LIN {X 0,Y 458.337,Z 1107.303,A -85,B 0,C 180,E1 22685.631,E2 22685.631} C_VEL
LIN {X 0,Y 458.982,Z 1103.583,A -85,B 0,C 180,E1 22683.619,E2 22683.619} C_VEL
LIN {X 0,Y 459.798,Z 1098.163,A -85,B 0,C 180,E1 22681.742,E2 22681.742} C_VEL
LIN {X 0,Y 460.852,Z 1090.743,A -85,B 0,C 180,E1 22679.873,E2 22679.873} C_VEL
LIN {X 0,Y 461.948,Z 1082.306,A -85,B 0,C 180,E1 22678.261,E2 22678.261} C_VEL
LIN {X 0,Y 463.216,Z 1071.686,A -85,B 0,C 180,E1 22676.656,E2 22676.656} C_VEL
LIN {X 0,Y 464.446,Z 1059.795,A -85,B 0,C 180,E1 22675.243,E2 22675.243} C_VEL
LIN {X 0,Y 465.635,Z 1046.257,A -85,B 0,C 180,E1 22673.958,E2 22673.958} C_VEL
LIN {X 0,Y 466.68,Z 1031.493,A -85,B 0,C 180,E1 22672.859,E2 22672.859} C_VEL
LIN {X 0,Y 467.361,Z 1018.628,A -85,B 0,C 180,E1 22672.128,E2 22672.128} C_VEL
LIN {X 0,Y 467.859,Z 1006.332,A -85,B 0,C 180,E1 22671.572,E2 22671.572} C_VEL
LIN {X 0,Y 468.216,Z 991.858,A -85,B 0,C 180,E1 22671.079,E2 22671.079} C_VEL
LIN {X 0,Y 469.132,Z 950.411,A -85,B 0,C 180,E1 22670.184,E2 22670.184} C_VEL
LIN {X 0,Y 473.462,Z 851.354,A -85,B 0,C 180,E1 22668.053,E2 22668.053} C_VEL
LIN {X 0,Y 475.333,Z 822.809,A -85,B 0,C 180,E1 22665.625,E2 22665.625} C_VEL
LIN {X 0,Y 478.095,Z 777.566,A -85,B 0,C 180,E1 22661.778,E2 22661.778} C_VEL
LIN {X 0,Y 480.688,Z 736.093,A -85,B 0,C 180,E1 22658.266,E2 22658.266} C_VEL
LIN {X 0,Y 483.225,Z 700.221,A -85,B 0,C 180,E1 22655.232,E2 22655.232} C_VEL
LIN {X 0,Y 479.813,Z 688.191,A -85,B 0,C 180,E1 22653.642,E2 22653.642} C_VEL
LIN {X 0,Y 475.221,Z 675.87,A -85,B 0,C 180,E1 22651.742,E2 22651.742} C_VEL
LIN {X 0,Y 470.89,Z 666.546,A -85,B 0,C 180,E1 22650.032,E2 22650.032} C_VEL
LIN {X 0,Y 467.066,Z 658.908,A -85,B 0,C 180,E1 22648.429,E2 22648.429} C_VEL
LIN {X 0,Y 464.878,Z 654.816,A -85,B 0,C 180,E1 22647.468,E2 22647.468} C_VEL
LIN {X 0,Y 462.283,Z 651.075,A -85,B 0,C 180,E1 22646.376,E2 22646.376} C_VEL
LIN {X 0,Y 461.646,Z 649.194,A -85,B 0,C 180,E1 22645.937,E2 22645.937} C_VEL
LIN {X 0,Y 458.957,Z 646.06,A -85,B 0,C 180,E1 22644.734,E2 22644.734} C_VEL
LIN {X 0,Y 458.216,Z 643.592,A -85,B 0,C 180,E1 22644.093,E2 22644.093} C_VEL
LIN {X 0,Y 458.23,Z 643.587,A -85,B 0,C 180,E1 22640.374,E2 22640.374} C_VEL
LIN {X 0,Y 458.266,Z 643.803,A -85,B 0,C 180,E1 22637.145,E2 22637.145} C_VEL
LIN {X 0,Y 465.849,Z 666.114,A -85,B 0,C 180,E1 22633.489,E2 22633.489} C_VEL
LIN {X 0,Y 468.816,Z 675.017,A -85,B 0,C 180,E1 22632.146,E2 22632.146} C_VEL
LIN {X 0,Y 486.171,Z 709.362,A -85,B 0,C 180,E1 22629.877,E2 22629.877} C_VEL
LIN {X 0,Y 491.258,Z 720.243,A -85,B 0,C 180,E1 22629.242,E2 22629.242} C_VEL
LIN {X 0,Y 494.064,Z 737.412,A -85,B 0,C 180,E1 22628.646,E2 22628.646} C_VEL
LIN {X 0,Y 482.629,Z 981.186,A -85,B 0,C 180,E1 22624.108,E2 22624.108} C_VEL
LIN {X 0,Y 480.802,Z 1004.838,A -85,B 0,C 180,E1 22623.453,E2 22623.453} C_VEL
LIN {X 0,Y 478.769,Z 1026.444,A -85,B 0,C 180,E1 22622.64,E2 22622.64} C_VEL
LIN {X 0,Y 476.333,Z 1048.657,A -85,B 0,C 180,E1 22621.581,E2 22621.581} C_VEL
LIN {X 0,Y 473.788,Z 1069.533,A -85,B 0,C 180,E1 22620.351,E2 22620.351} C_VEL
LIN {X 0,Y 471.164,Z 1089.497,A -85,B 0,C 180,E1 22618.935,E2 22618.935} C_VEL
LIN {X 0,Y 468.474,Z 1108.558,A -85,B 0,C 180,E1 22617.313,E2 22617.313} C_VEL
LIN {X 0,Y 465.955,Z 1126.145,A -85,B 0,C 180,E1 22615.549,E2 22615.549} C_VEL
LIN {X 0,Y 463.62,Z 1142.393,A -85,B 0,C 180,E1 22613.648,E2 22613.648} C_VEL
LIN {X 0,Y 461.556,Z 1157.308,A -85,B 0,C 180,E1 22611.607,E2 22611.607} C_VEL
LIN {X 0,Y 459.786,Z 1170.792,A -85,B 0,C 180,E1 22609.432,E2 22609.432} C_VEL
LIN {X 0,Y 458.295,Z 1183.586,A -85,B 0,C 180,E1 22606.997,E2 22606.997} C_VEL
LIN {X 0,Y 457.241,Z 1194.282,A -85,B 0,C 180,E1 22604.563,E2 22604.563} C_VEL
LIN {X 0,Y 456.575,Z 1203.017,A -85,B 0,C 180,E1 22602.134,E2 22602.134} C_VEL
LIN {X 0,Y 456.199,Z 1210.324,A -85,B 0,C 180,E1 22599.587,E2 22599.587} C_VEL
LIN {X 0,Y 456.065,Z 1215.915,A -85,B 0,C 180,E1 22597.05,E2 22597.05} C_VEL
LIN {X 0,Y 456.056,Z 1219.591,A -85,B 0,C 180,E1 22594.651,E2 22594.651} C_VEL
LIN {X 0,Y 456.097,Z 1221.978,A -85,B 0,C 180,E1 22592.008,E2 22592.008} C_VEL
LIN {X 0,Y 456.094,Z 1222.654,A -85,B 0,C 180,E1 22589.621,E2 22589.621} C_VEL
LIN {X 0,Y 456.059,Z 1221.739,A -85,B 0,C 180,E1 22587.108,E2 22587.108} C_VEL
LIN {X 0,Y 456.022,Z 1219.335,A -85,B 0,C 180,E1 22584.588,E2 22584.588} C_VEL
LIN {X 0,Y 456.064,Z 1215.225,A -85,B 0,C 180,E1 22582.059,E2 22582.059} C_VEL
LIN {X 0,Y 456.309,Z 1209.17,A -85,B 0,C 180,E1 22579.392,E2 22579.392} C_VEL
LIN {X 0,Y 456.847,Z 1201.683,A -85,B 0,C 180,E1 22576.841,E2 22576.841} C_VEL
LIN {X 0,Y 457.781,Z 1192.207,A -85,B 0,C 180,E1 22574.284,E2 22574.284} C_VEL
LIN {X 0,Y 459.122,Z 1181.351,A -85,B 0,C 180,E1 22571.853,E2 22571.853} C_VEL
LIN {X 0,Y 460.874,Z 1169.238,A -85,B 0,C 180,E1 22569.554,E2 22569.554} C_VEL
LIN {X 0,Y 463.122,Z 1154.921,A -85,B 0,C 180,E1 22567.264,E2 22567.264} C_VEL
LIN {X 0,Y 465.787,Z 1139.175,A -85,B 0,C 180,E1 22565.117,E2 22565.117} C_VEL
LIN {X 0,Y 468.983,Z 1120.873,A -85,B 0,C 180,E1 22562.99,E2 22562.99} C_VEL
LIN {X 0,Y 472.427,Z 1101.443,A -85,B 0,C 180,E1 22561.081,E2 22561.081} C_VEL
LIN {X 0,Y 475.913,Z 1081.805,A -85,B 0,C 180,E1 22559.439,E2 22559.439} C_VEL
LIN {X 0,Y 479.703,Z 1059.729,A -85,B 0,C 180,E1 22557.89,E2 22557.89} C_VEL
LIN {X 0,Y 483.529,Z 1036.671,A -85,B 0,C 180,E1 22556.556,E2 22556.556} C_VEL
LIN {X 0,Y 487.071,Z 1014.04,A -85,B 0,C 180,E1 22555.486,E2 22555.486} C_VEL
LIN {X 0,Y 490.729,Z 988.982,A -85,B 0,C 180,E1 22554.548,E2 22554.548} C_VEL
LIN {X 0,Y 494.01,Z 962.501,A -85,B 0,C 180,E1 22553.788,E2 22553.788} C_VEL
LIN {X 0,Y 502.512,Z 886.864,A -85,B 0,C 180,E1 22551.886,E2 22551.886} C_VEL
LIN {X 0,Y 512.742,Z 815.166,A -85,B 0,C 180,E1 22550.007,E2 22550.007} C_VEL
LIN {X 0,Y 525.324,Z 742.891,A -85,B 0,C 180,E1 22548.094,E2 22548.094} C_VEL
LIN {X 0,Y 525.625,Z 739.764,A -85,B 0,C 180,E1 22547.895,E2 22547.895} C_VEL
LIN {X 0,Y 524.85,Z 735.088,A -85,B 0,C 180,E1 22546.983,E2 22546.983} C_VEL
LIN {X 0,Y 524.367,Z 731.897,A -85,B 0,C 180,E1 22546.122,E2 22546.122} C_VEL
LIN {X 0,Y 524.118,Z 729.55,A -85,B 0,C 180,E1 22545.057,E2 22545.057} C_VEL
LIN {X 0,Y 524.379,Z 728.32,A -85,B 0,C 180,E1 22544.038,E2 22544.038} C_VEL
LIN {X 0,Y 525.489,Z 728.89,A -85,B 0,C 180,E1 22542.575,E2 22542.575} C_VEL
LIN {X 0,Y 526.895,Z 731.802,A -85,B 0,C 180,E1 22541.405,E2 22541.405} C_VEL
LIN {X 0,Y 513.622,Z 804.551,A -85,B 0,C 180,E1 22539.481,E2 22539.481} C_VEL
LIN {X 0,Y 503.47,Z 872.417,A -85,B 0,C 180,E1 22537.696,E2 22537.696} C_VEL
LIN {X 0,Y 494.22,Z 950.824,A -85,B 0,C 180,E1 22535.659,E2 22535.659} C_VEL
LIN {X 0,Y 491.286,Z 974.469,A -85,B 0,C 180,E1 22534.814,E2 22534.814} C_VEL
LIN {X 0,Y 488.112,Z 997.009,A -85,B 0,C 180,E1 22533.793,E2 22533.793} C_VEL
LIN {X 0,Y 484.564,Z 1019.669,A -85,B 0,C 180,E1 22532.518,E2 22532.518} C_VEL
LIN {X 0,Y 480.93,Z 1040.911,A -85,B 0,C 180,E1 22531.064,E2 22531.064} C_VEL
LIN {X 0,Y 477.15,Z 1061.537,A -85,B 0,C 180,E1 22529.366,E2 22529.366} C_VEL
LIN {X 0,Y 473.79,Z 1078.913,A -85,B 0,C 180,E1 22527.667,E2 22527.667} C_VEL
LIN {X 0,Y 470.383,Z 1096.053,A -85,B 0,C 180,E1 22525.701,E2 22525.701} C_VEL
LIN {X 0,Y 467.258,Z 1111.645,A -85,B 0,C 180,E1 22523.591,E2 22523.591} C_VEL
LIN {X 0,Y 464.455,Z 1125.746,A -85,B 0,C 180,E1 22521.338,E2 22521.338} C_VEL
LIN {X 0,Y 462.024,Z 1138.267,A -85,B 0,C 180,E1 22518.945,E2 22518.945} C_VEL
LIN {X 0,Y 460.099,Z 1148.714,A -85,B 0,C 180,E1 22516.543,E2 22516.543} C_VEL
LIN {X 0,Y 458.529,Z 1158.219,A -85,B 0,C 180,E1 22513.881,E2 22513.881} C_VEL
LIN {X 0,Y 457.491,Z 1165.473,A -85,B 0,C 180,E1 22511.347,E2 22511.347} C_VEL
LIN {X 0,Y 456.811,Z 1170.96,A -85,B 0,C 180,E1 22508.816,E2 22508.816} C_VEL
LIN {X 0,Y 456.398,Z 1175.063,A -85,B 0,C 180,E1 22506.165,E2 22506.165} C_VEL
LIN {X 0,Y 456.205,Z 1177.569,A -85,B 0,C 180,E1 22503.521,E2 22503.521} C_VEL
LIN {X 0,Y 456.123,Z 1178.354,A -85,B 0,C 180,E1 22501.008,E2 22501.008} C_VEL
LIN {X 0,Y 456.09,Z 1177.621,A -85,B 0,C 180,E1 22498.37,E2 22498.37} C_VEL
LIN {X 0,Y 456.122,Z 1175.459,A -85,B 0,C 180,E1 22495.854,E2 22495.854} C_VEL
LIN {X 0,Y 456.255,Z 1171.659,A -85,B 0,C 180,E1 22493.333,E2 22493.333} C_VEL
LIN {X 0,Y 456.568,Z 1166.024,A -85,B 0,C 180,E1 22490.676,E2 22490.676} C_VEL
LIN {X 0,Y 457.13,Z 1158.966,A -85,B 0,C 180,E1 22488.138,E2 22488.138} C_VEL
LIN {X 0,Y 458.014,Z 1149.951,A -85,B 0,C 180,E1 22485.592,E2 22485.592} C_VEL
LIN {X 0,Y 459.234,Z 1139.531,A -85,B 0,C 180,E1 22483.17,E2 22483.17} C_VEL
LIN {X 0,Y 460.786,Z 1127.797,A -85,B 0,C 180,E1 22480.876,E2 22480.876} C_VEL
LIN {X 0,Y 462.67,Z 1114.375,A -85,B 0,C 180,E1 22478.664,E2 22478.664} C_VEL
LIN {X 0,Y 464.862,Z 1099.284,A -85,B 0,C 180,E1 22476.555,E2 22476.555} C_VEL
LIN {X 0,Y 467.373,Z 1082.277,A -85,B 0,C 180,E1 22474.533,E2 22474.533} C_VEL
LIN {X 0,Y 469.879,Z 1064.944,A -85,B 0,C 180,E1 22472.777,E2 22472.777} C_VEL
LIN {X 0,Y 472.502,Z 1046.063,A -85,B 0,C 180,E1 22471.156,E2 22471.156} C_VEL
LIN {X 0,Y 475.044,Z 1025.969,A -85,B 0,C 180,E1 22469.713,E2 22469.713} C_VEL
LIN {X 0,Y 477.5,Z 1004.905,A -85,B 0,C 180,E1 22468.46,E2 22468.46} C_VEL
LIN {X 0,Y 479.725,Z 983.049,A -85,B 0,C 180,E1 22467.402,E2 22467.402} C_VEL
LIN {X 0,Y 481.61,Z 960.789,A -85,B 0,C 180,E1 22466.551,E2 22466.551} C_VEL
LIN {X 0,Y 483.181,Z 937.605,A -85,B 0,C 180,E1 22465.897,E2 22465.897} C_VEL
LIN {X 0,Y 485.692,Z 881.128,A -85,B 0,C 180,E1 22464.823,E2 22464.823} C_VEL
LIN {X 0,Y 493.87,Z 706.895,A -85,B 0,C 180,E1 22461.609,E2 22461.609} C_VEL
LIN {X 0,Y 473.868,Z 671.342,A -85,B 0,C 180,E1 22459.2,E2 22459.2} C_VEL
LIN {X 0,Y 459.932,Z 647.609,A -85,B 0,C 180,E1 22457.384,E2 22457.384} C_VEL
LIN {X 0,Y 458.349,Z 644.303,A -85,B 0,C 180,E1 22457.157,E2 22457.157} C_VEL
LIN {X 0,Y 458.226,Z 643.591,A -85,B 0,C 180,E1 22457.098,E2 22457.098} C_VEL
LIN {X 0,Y 458.204,Z 643.595,A -85,B 0,C 180,E1 22453.397,E2 22453.397} C_VEL
LIN {X 0,Y 458.194,Z 643.592,A -85,B 0,C 180,E1 22449.818,E2 22449.818} C_VEL
LIN {X 0,Y 458.229,Z 643.588,A -85,B 0,C 180,E1 22446.099,E2 22446.099} C_VEL
LIN {X 0,Y 458.238,Z 643.584,A -85,B 0,C 180,E1 22442.394,E2 22442.394} C_VEL
LIN {X 0,Y 458.226,Z 643.59,A -85,B 0,C 180,E1 22438.691,E2 22438.691} C_VEL
LIN {X 0,Y 458.208,Z 643.593,A -85,B 0,C 180,E1 22435.047,E2 22435.047} C_VEL
LIN {X 0,Y 458.209,Z 643.589,A -85,B 0,C 180,E1 22431.508,E2 22431.508} C_VEL
LIN {X 0,Y 458.228,Z 643.582,A -85,B 0,C 180,E1 22427.789,E2 22427.789} C_VEL
LIN {X 0,Y 458.24,Z 643.579,A -85,B 0,C 180,E1 22424.147,E2 22424.147} C_VEL
LIN {X 0,Y 458.227,Z 643.59,A -85,B 0,C 180,E1 22420.436,E2 22420.436} C_VEL
LIN {X 0,Y 458.221,Z 643.588,A -85,B 0,C 180,E1 22416.769,E2 22416.769} C_VEL
LIN {X 0,Y 458.199,Z 643.579,A -85,B 0,C 180,E1 22413.004,E2 22413.004} C_VEL
LIN {X 0,Y 458.243,Z 643.589,A -85,B 0,C 180,E1 22409.252,E2 22409.252} C_VEL
LIN {X 0,Y 458.23,Z 643.574,A -85,B 0,C 180,E1 22405.496,E2 22405.496} C_VEL
LIN {X 0,Y 458.241,Z 643.586,A -85,B 0,C 180,E1 22402.552,E2 22402.552} C_VEL
LIN {X 0,Y 457.257,Z 643.71,A -85,B 0,C 180,E1 22401.59,E2 22401.59} C_VEL
LIN {X 0,Y 450.741,Z 644.5,A -85,B 0,C 180,E1 22398.81,E2 22398.81} C_VEL
LIN {X 0,Y 450.263,Z 644.562,A -85,B 0,C 180,E1 22398.173,E2 22398.173} C_VEL
LIN {X 0,Y 450.272,Z 644.581,A -85,B 0,C 180,E1 22394.512,E2 22394.512} C_VEL
LIN {X 0,Y 450.297,Z 644.578,A -85,B 0,C 180,E1 22390.816,E2 22390.816} C_VEL
LIN {X 0,Y 450.3,Z 644.576,A -85,B 0,C 180,E1 22387.136,E2 22387.136} C_VEL
LIN {X 0,Y 450.282,Z 644.581,A -85,B 0,C 180,E1 22383.351,E2 22383.351} C_VEL
LIN {X 0,Y 450.266,Z 644.582,A -85,B 0,C 180,E1 22379.732,E2 22379.732} C_VEL
LIN {X 0,Y 450.271,Z 644.582,A -85,B 0,C 180,E1 22375.975,E2 22375.975} C_VEL
LIN {X 0,Y 450.303,Z 644.577,A -85,B 0,C 180,E1 22372.207,E2 22372.207} C_VEL
LIN {X 0,Y 450.293,Z 644.577,A -85,B 0,C 180,E1 22368.439,E2 22368.439} C_VEL
LIN {X 0,Y 450.313,Z 644.69,A -85,B 0,C 180,E1 22367.619,E2 22367.619} C_VEL
LIN {X 0,Y 458.281,Z 670.797,A -85,B 0,C 180,E1 22364.754,E2 22364.754} C_VEL
LIN {X 0,Y 463.683,Z 690.602,A -85,B 0,C 180,E1 22362.668,E2 22362.668} C_VEL
LIN {X 0,Y 461.849,Z 733.114,A -85,B 0,C 180,E1 22358.997,E2 22358.997} C_VEL
LIN {X 0,Y 460.019,Z 774.082,A -85,B 0,C 180,E1 22355.471,E2 22355.471} C_VEL
LIN {X 0,Y 458.233,Z 816.759,A -85,B 0,C 180,E1 22351.8,E2 22351.8} C_VEL
LIN {X 0,Y 457.335,Z 841.237,A -85,B 0,C 180,E1 22349.747,E2 22349.747} C_VEL
LIN {X 0,Y 454.489,Z 984.58,A -85,B 0,C 180,E1 22346.943,E2 22346.943} C_VEL
LIN {X 0,Y 454.254,Z 1000.505,A -85,B 0,C 180,E1 22346.432,E2 22346.432} C_VEL
LIN {X 0,Y 453.773,Z 1017.239,A -85,B 0,C 180,E1 22345.654,E2 22345.654} C_VEL
LIN {X 0,Y 453.21,Z 1032.259,A -85,B 0,C 180,E1 22344.71,E2 22344.71} C_VEL
LIN {X 0,Y 452.517,Z 1047.114,A -85,B 0,C 180,E1 22343.516,E2 22343.516} C_VEL
LIN {X 0,Y 451.77,Z 1060.968,A -85,B 0,C 180,E1 22342.099,E2 22342.099} C_VEL
LIN {X 0,Y 451.111,Z 1072.473,A -85,B 0,C 180,E1 22340.632,E2 22340.632} C_VEL
LIN {X 0,Y 450.49,Z 1083.338,A -85,B 0,C 180,E1 22338.905,E2 22338.905} C_VEL
LIN {X 0,Y 450.048,Z 1091.85,A -85,B 0,C 180,E1 22337.184,E2 22337.184} C_VEL
LIN {X 0,Y 449.732,Z 1099.321,A -85,B 0,C 180,E1 22335.233,E2 22335.233} C_VEL
LIN {X 0,Y 449.564,Z 1104.421,A -85,B 0,C 180,E1 22333.371,E2 22333.371} C_VEL
LIN {X 0,Y 449.564,Z 1108.099,A -85,B 0,C 180,E1 22331.414,E2 22331.414} C_VEL
LIN {X 0,Y 449.693,Z 1109.939,A -85,B 0,C 180,E1 22329.467,E2 22329.467} C_VEL
LIN {X 0,Y 450.004,Z 1110.041,A -85,B 0,C 180,E1 22327.402,E2 22327.402} C_VEL
LIN {X 0,Y 450.468,Z 1108.36,A -85,B 0,C 180,E1 22325.474,E2 22325.474} C_VEL
LIN {X 0,Y 451.167,Z 1104.684,A -85,B 0,C 180,E1 22323.428,E2 22323.428} C_VEL
LIN {X 0,Y 452.05,Z 1099.312,A -85,B 0,C 180,E1 22321.518,E2 22321.518} C_VEL
LIN {X 0,Y 453.175,Z 1091.901,A -85,B 0,C 180,E1 22319.618,E2 22319.618} C_VEL
LIN {X 0,Y 454.34,Z 1083.471,A -85,B 0,C 180,E1 22317.979,E2 22317.979} C_VEL
LIN {X 0,Y 455.686,Z 1072.872,A -85,B 0,C 180,E1 22316.349,E2 22316.349} C_VEL
LIN {X 0,Y 457.004,Z 1061.08,A -85,B 0,C 180,E1 22314.914,E2 22314.914} C_VEL
LIN {X 0,Y 458.218,Z 1048.37,A -85,B 0,C 180,E1 22313.671,E2 22313.671} C_VEL
LIN {X 0,Y 459.312,Z 1033.812,A -85,B 0,C 180,E1 22312.555,E2 22312.555} C_VEL
LIN {X 0,Y 460.035,Z 1021.306,A -85,B 0,C 180,E1 22311.813,E2 22311.813} C_VEL
LIN {X 0,Y 460.598,Z 1008.702,A -85,B 0,C 180,E1 22311.218,E2 22311.218} C_VEL
LIN {X 0,Y 461.027,Z 993.799,A -85,B 0,C 180,E1 22310.685,E2 22310.685} C_VEL
LIN {X 0,Y 461.915,Z 955.217,A -85,B 0,C 180,E1 22309.813,E2 22309.813} C_VEL
LIN {X 0,Y 466.569,Z 853.052,A -85,B 0,C 180,E1 22307.576,E2 22307.576} C_VEL
LIN {X 0,Y 467.129,Z 848.404,A -85,B 0,C 180,E1 22307.198,E2 22307.198} C_VEL
LIN {X 0,Y 470.047,Z 802.606,A -85,B 0,C 180,E1 22303.245,E2 22303.245} C_VEL
LIN {X 0,Y 472.898,Z 759.889,A -85,B 0,C 180,E1 22299.579,E2 22299.579} C_VEL
LIN {X 0,Y 476.042,Z 716.875,A -85,B 0,C 180,E1 22295.885,E2 22295.885} C_VEL
LIN {X 0,Y 477.044,Z 703.66,A -85,B 0,C 180,E1 22294.75,E2 22294.75} C_VEL
LIN {X 0,Y 473.589,Z 691.406,A -85,B 0,C 180,E1 22293.063,E2 22293.063} C_VEL
LIN {X 0,Y 469.425,Z 680.099,A -85,B 0,C 180,E1 22291.222,E2 22291.222} C_VEL
LIN {X 0,Y 464.623,Z 669.452,A -85,B 0,C 180,E1 22289.162,E2 22289.162} C_VEL
LIN {X 0,Y 462.016,Z 664.602,A -85,B 0,C 180,E1 22288.029,E2 22288.029} C_VEL
LIN {X 0,Y 459.954,Z 660.63,A -85,B 0,C 180,E1 22287.043,E2 22287.043} C_VEL
LIN {X 0,Y 457.831,Z 657.042,A -85,B 0,C 180,E1 22286.004,E2 22286.004} C_VEL
LIN {X 0,Y 457.236,Z 655.752,A -85,B 0,C 180,E1 22285.651,E2 22285.651} C_VEL
LIN {X 0,Y 454.733,Z 652.236,A -85,B 0,C 180,E1 22284.357,E2 22284.357} C_VEL
LIN {X 0,Y 454.056,Z 650.421,A -85,B 0,C 180,E1 22283.828,E2 22283.828} C_VEL
LIN {X 0,Y 451.212,Z 647.452,A -85,B 0,C 180,E1 22282.13,E2 22282.13} C_VEL
LIN {X 0,Y 450.294,Z 644.579,A -85,B 0,C 180,E1 22281,E2 22281} C_VEL
LIN {X 0,Y 450.298,Z 644.624,A -85,B 0,C 180,E1 22277.807,E2 22277.807} C_VEL
LIN {X 0,Y 457.888,Z 666.977,A -85,B 0,C 180,E1 22274.072,E2 22274.072} C_VEL
LIN {X 0,Y 460.437,Z 674.616,A -85,B 0,C 180,E1 22272.889,E2 22272.889} C_VEL
LIN {X 0,Y 477.823,Z 708.748,A -85,B 0,C 180,E1 22270.568,E2 22270.568} C_VEL
LIN {X 0,Y 484.83,Z 723.669,A -85,B 0,C 180,E1 22269.653,E2 22269.653} C_VEL
LIN {X 0,Y 487.245,Z 738.83,A -85,B 0,C 180,E1 22269.123,E2 22269.123} C_VEL
LIN {X 0,Y 475.415,Z 980.893,A -85,B 0,C 180,E1 22264.525,E2 22264.525} C_VEL
LIN {X 0,Y 473.536,Z 1004.519,A -85,B 0,C 180,E1 22263.86,E2 22263.86} C_VEL
LIN {X 0,Y 471.377,Z 1026.768,A -85,B 0,C 180,E1 22263.007,E2 22263.007} C_VEL
LIN {X 0,Y 468.865,Z 1048.922,A -85,B 0,C 180,E1 22261.927,E2 22261.927} C_VEL
LIN {X 0,Y 466.265,Z 1069.575,A -85,B 0,C 180,E1 22260.687,E2 22260.687} C_VEL
LIN {X 0,Y 463.558,Z 1089.559,A -85,B 0,C 180,E1 22259.243,E2 22259.243} C_VEL
LIN {X 0,Y 460.796,Z 1108.578,A -85,B 0,C 180,E1 22257.596,E2 22257.596} C_VEL
LIN {X 0,Y 458.208,Z 1126.129,A -85,B 0,C 180,E1 22255.805,E2 22255.805} C_VEL
LIN {X 0,Y 455.729,Z 1142.879,A -85,B 0,C 180,E1 22253.802,E2 22253.802} C_VEL
LIN {X 0,Y 453.626,Z 1157.705,A -85,B 0,C 180,E1 22251.732,E2 22251.732} C_VEL
LIN {X 0,Y 451.778,Z 1171.427,A -85,B 0,C 180,E1 22249.462,E2 22249.462} C_VEL
LIN {X 0,Y 450.301,Z 1183.795,A -85,B 0,C 180,E1 22247.042,E2 22247.042} C_VEL
LIN {X 0,Y 449.235,Z 1194.392,A -85,B 0,C 180,E1 22244.565,E2 22244.565} C_VEL
LIN {X 0,Y 448.564,Z 1203.082,A -85,B 0,C 180,E1 22242.093,E2 22242.093} C_VEL
LIN {X 0,Y 448.202,Z 1210.109,A -85,B 0,C 180,E1 22239.571,E2 22239.571} C_VEL
LIN {X 0,Y 448.073,Z 1215.549,A -85,B 0,C 180,E1 22237.048,E2 22237.048} C_VEL
LIN {X 0,Y 448.068,Z 1219.215,A -85,B 0,C 180,E1 22234.606,E2 22234.606} C_VEL
LIN {X 0,Y 448.11,Z 1221.575,A -85,B 0,C 180,E1 22231.916,E2 22231.916} C_VEL
LIN {X 0,Y 448.104,Z 1222.229,A -85,B 0,C 180,E1 22229.487,E2 22229.487} C_VEL
LIN {X 0,Y 448.062,Z 1221.271,A -85,B 0,C 180,E1 22226.928,E2 22226.928} C_VEL
LIN {X 0,Y 448.023,Z 1218.823,A -85,B 0,C 180,E1 22224.363,E2 22224.363} C_VEL
LIN {X 0,Y 448.083,Z 1214.671,A -85,B 0,C 180,E1 22221.788,E2 22221.788} C_VEL
LIN {X 0,Y 448.361,Z 1208.565,A -85,B 0,C 180,E1 22219.071,E2 22219.071} C_VEL
LIN {X 0,Y 448.964,Z 1201.029,A -85,B 0,C 180,E1 22216.475,E2 22216.475} C_VEL
LIN {X 0,Y 449.989,Z 1191.515,A -85,B 0,C 180,E1 22213.872,E2 22213.872} C_VEL
LIN {X 0,Y 451.451,Z 1180.617,A -85,B 0,C 180,E1 22211.4,E2 22211.4} C_VEL
LIN {X 0,Y 453.468,Z 1167.711,A -85,B 0,C 180,E1 22208.934,E2 22208.934} C_VEL
LIN {X 0,Y 455.924,Z 1153.321,A -85,B 0,C 180,E1 22206.611,E2 22206.611} C_VEL
LIN {X 0,Y 458.888,Z 1136.937,A -85,B 0,C 180,E1 22204.371,E2 22204.371} C_VEL
LIN {X 0,Y 462.147,Z 1119.572,A -85,B 0,C 180,E1 22202.347,E2 22202.347} C_VEL
LIN {X 0,Y 465.834,Z 1100.126,A -85,B 0,C 180,E1 22200.416,E2 22200.416} C_VEL
LIN {X 0,Y 469.684,Z 1079.787,A -85,B 0,C 180,E1 22198.704,E2 22198.704} C_VEL
LIN {X 0,Y 473.774,Z 1057.66,A -85,B 0,C 180,E1 22197.14,E2 22197.14} C_VEL
LIN {X 0,Y 478.026,Z 1033.867,A -85,B 0,C 180,E1 22195.758,E2 22195.758} C_VEL
LIN {X 0,Y 482.157,Z 1009.227,A -85,B 0,C 180,E1 22194.601,E2 22194.601} C_VEL
LIN {X 0,Y 486.308,Z 982.698,A -85,B 0,C 180,E1 22193.639,E2 22193.639} C_VEL
LIN {X 0,Y 490.024,Z 953.283,A -85,B 0,C 180,E1 22192.82,E2 22192.82} C_VEL
LIN {X 0,Y 498.645,Z 884.788,A -85,B 0,C 180,E1 22191.04,E2 22191.04} C_VEL
LIN {X 0,Y 509.832,Z 813.836,A -85,B 0,C 180,E1 22189.136,E2 22189.136} C_VEL
LIN {X 0,Y 522.832,Z 745.199,A -85,B 0,C 180,E1 22187.29,E2 22187.29} C_VEL
LIN {X 0,Y 522.275,Z 739.861,A -85,B 0,C 180,E1 22186.088,E2 22186.088} C_VEL
LIN {X 0,Y 522.1,Z 737.122,A -85,B 0,C 180,E1 22184.878,E2 22184.878} C_VEL
LIN {X 0,Y 522.417,Z 736.065,A -85,B 0,C 180,E1 22183.973,E2 22183.973} C_VEL
LIN {X 0,Y 523.403,Z 736.623,A -85,B 0,C 180,E1 22182.65,E2 22182.65} C_VEL
LIN {X 0,Y 523.881,Z 737.963,A -85,B 0,C 180,E1 22182.109,E2 22182.109} C_VEL
LIN {X 0,Y 509.719,Z 810.287,A -85,B 0,C 180,E1 22180.174,E2 22180.174} C_VEL
LIN {X 0,Y 498.675,Z 878.354,A -85,B 0,C 180,E1 22178.342,E2 22178.342} C_VEL
LIN {X 0,Y 489.185,Z 951.63,A -85,B 0,C 180,E1 22176.378,E2 22176.378} C_VEL
LIN {X 0,Y 486.052,Z 974.778,A -85,B 0,C 180,E1 22175.534,E2 22175.534} C_VEL
LIN {X 0,Y 482.482,Z 997.964,A -85,B 0,C 180,E1 22174.457,E2 22174.457} C_VEL
LIN {X 0,Y 478.713,Z 1020.215,A -85,B 0,C 180,E1 22173.18,E2 22173.18} C_VEL
LIN {X 0,Y 474.796,Z 1041.439,A -85,B 0,C 180,E1 22171.7,E2 22171.7} C_VEL
LIN {X 0,Y 470.962,Z 1060.961,A -85,B 0,C 180,E1 22170.072,E2 22170.072} C_VEL
LIN {X 0,Y 467.253,Z 1078.976,A -85,B 0,C 180,E1 22168.296,E2 22168.296} C_VEL
LIN {X 0,Y 463.519,Z 1096.576,A -85,B 0,C 180,E1 22166.248,E2 22166.248} C_VEL
LIN {X 0,Y 460.252,Z 1111.837,A -85,B 0,C 180,E1 22164.153,E2 22164.153} C_VEL
LIN {X 0,Y 457.35,Z 1125.463,A -85,B 0,C 180,E1 22161.956,E2 22161.956} C_VEL
LIN {X 0,Y 454.706,Z 1138.037,A -85,B 0,C 180,E1 22159.529,E2 22159.529} C_VEL
LIN {X 0,Y 452.617,Z 1148.6,A -85,B 0,C 180,E1 22157.089,E2 22157.089} C_VEL
LIN {X 0,Y 450.951,Z 1157.821,A -85,B 0,C 180,E1 22154.513,E2 22154.513} C_VEL
LIN {X 0,Y 449.713,Z 1165.568,A -85,B 0,C 180,E1 22151.806,E2 22151.806} C_VEL
LIN {X 0,Y 448.912,Z 1171.367,A -85,B 0,C 180,E1 22149.102,E2 22149.102} C_VEL
LIN {X 0,Y 448.452,Z 1175.481,A -85,B 0,C 180,E1 22146.403,E2 22146.403} C_VEL
LIN {X 0,Y 448.235,Z 1177.933,A -85,B 0,C 180,E1 22143.84,E2 22143.84} C_VEL
LIN {X 0,Y 448.138,Z 1178.782,A -85,B 0,C 180,E1 22141.153,E2 22141.153} C_VEL
LIN {X 0,Y 448.1,Z 1178.058,A -85,B 0,C 180,E1 22138.468,E2 22138.468} C_VEL
LIN {X 0,Y 448.13,Z 1175.827,A -85,B 0,C 180,E1 22135.852,E2 22135.852} C_VEL
LIN {X 0,Y 448.263,Z 1172.08,A -85,B 0,C 180,E1 22133.342,E2 22133.342} C_VEL
LIN {X 0,Y 448.584,Z 1166.432,A -85,B 0,C 180,E1 22130.638,E2 22130.638} C_VEL
LIN {X 0,Y 449.164,Z 1159.356,A -85,B 0,C 180,E1 22128.055,E2 22128.055} C_VEL
LIN {X 0,Y 450.077,Z 1150.31,A -85,B 0,C 180,E1 22125.464,E2 22125.464} C_VEL
LIN {X 0,Y 451.34,Z 1139.852,A -85,B 0,C 180,E1 22123,E2 22123} C_VEL
LIN {X 0,Y 452.946,Z 1128.076,A -85,B 0,C 180,E1 22120.666,E2 22120.666} C_VEL
LIN {X 0,Y 454.915,Z 1114.487,A -85,B 0,C 180,E1 22118.397,E2 22118.397} C_VEL
LIN {X 0,Y 457.161,Z 1099.458,A -85,B 0,C 180,E1 22116.273,E2 22116.273} C_VEL
LIN {X 0,Y 459.765,Z 1082.277,A -85,B 0,C 180,E1 22114.207,E2 22114.207} C_VEL
LIN {X 0,Y 462.434,Z 1064.263,A -85,B 0,C 180,E1 22112.371,E2 22112.371} C_VEL
LIN {X 0,Y 465.146,Z 1045.216,A -85,B 0,C 180,E1 22110.726,E2 22110.726} C_VEL
LIN {X 0,Y 467.753,Z 1025.162,A -85,B 0,C 180,E1 22109.28,E2 22109.28} C_VEL
LIN {X 0,Y 470.234,Z 1004.3,A -85,B 0,C 180,E1 22108.035,E2 22108.035} C_VEL
LIN {X 0,Y 472.542,Z 981.975,A -85,B 0,C 180,E1 22106.952,E2 22106.952} C_VEL
LIN {X 0,Y 474.47,Z 959.621,A -85,B 0,C 180,E1 22106.1,E2 22106.1} C_VEL
LIN {X 0,Y 476.08,Z 936.494,A -85,B 0,C 180,E1 22105.446,E2 22105.446} C_VEL
LIN {X 0,Y 486.993,Z 709.745,A -85,B 0,C 180,E1 22101.155,E2 22101.155} C_VEL
LIN {X 0,Y 468.252,Z 676.264,A -85,B 0,C 180,E1 22098.851,E2 22098.851} C_VEL
LIN {X 0,Y 454.07,Z 652.183,A -85,B 0,C 180,E1 22096.979,E2 22096.979} C_VEL
LIN {X 0,Y 451.858,Z 648.432,A -85,B 0,C 180,E1 22096.676,E2 22096.676} C_VEL
LIN {X 0,Y 450.372,Z 645.082,A -85,B 0,C 180,E1 22096.448,E2 22096.448} C_VEL
LIN {X 0,Y 450.293,Z 644.574,A -85,B 0,C 180,E1 22096.424,E2 22096.424} C_VEL
LIN {X 0,Y 450.252,Z 644.581,A -85,B 0,C 180,E1 22092.81,E2 22092.81} C_VEL
LIN {X 0,Y 450.22,Z 644.588,A -85,B 0,C 180,E1 22089.106,E2 22089.106} C_VEL
LIN {X 0,Y 450.257,Z 644.576,A -85,B 0,C 180,E1 22085.419,E2 22085.419} C_VEL
LIN {X 0,Y 450.293,Z 644.576,A -85,B 0,C 180,E1 22081.745,E2 22081.745} C_VEL
LIN {X 0,Y 450.287,Z 644.58,A -85,B 0,C 180,E1 22078.085,E2 22078.085} C_VEL
LIN {X 0,Y 450.247,Z 644.585,A -85,B 0,C 180,E1 22074.399,E2 22074.399} C_VEL
LIN {X 0,Y 450.222,Z 644.586,A -85,B 0,C 180,E1 22070.68,E2 22070.68} C_VEL
LIN {X 0,Y 450.264,Z 644.577,A -85,B 0,C 180,E1 22067.047,E2 22067.047} C_VEL
LIN {X 0,Y 450.299,Z 644.564,A -85,B 0,C 180,E1 22063.466,E2 22063.466} C_VEL
LIN {X 0,Y 450.276,Z 644.574,A -85,B 0,C 180,E1 22059.718,E2 22059.718} C_VEL
LIN {X 0,Y 450.239,Z 644.583,A -85,B 0,C 180,E1 22055.993,E2 22055.993} C_VEL
LIN {X 0,Y 450.222,Z 644.571,A -85,B 0,C 180,E1 22052.102,E2 22052.102} C_VEL
LIN {X 0,Y 450.264,Z 644.578,A -85,B 0,C 180,E1 22048.475,E2 22048.475} C_VEL
LIN {X 0,Y 450.294,Z 644.566,A -85,B 0,C 180,E1 22044.778,E2 22044.778} C_VEL
LIN {X 0,Y 450.274,Z 644.574,A -85,B 0,C 180,E1 22041.155,E2 22041.155} C_VEL
LIN {X 0,Y 450.263,Z 644.562,A -85,B 0,C 180,E1 22038.173,E2 22038.173} C_VEL
LIN {X 0,Y 449.22,Z 644.701,A -85,B 0,C 180,E1 22037.193,E2 22037.193} C_VEL
LIN {X 0,Y 442.721,Z 645.52,A -85,B 0,C 180,E1 22034.363,E2 22034.363} C_VEL
LIN {X 0,Y 442.29,Z 645.57,A -85,B 0,C 180,E1 22033.715,E2 22033.715} C_VEL
LIN {X 0,Y 442.334,Z 645.565,A -85,B 0,C 180,E1 22030.044,E2 22030.044} C_VEL
LIN {X 0,Y 442.361,Z 645.561,A -85,B 0,C 180,E1 22026.419,E2 22026.419} C_VEL
LIN {X 0,Y 442.334,Z 645.567,A -85,B 0,C 180,E1 22022.661,E2 22022.661} C_VEL
LIN {X 0,Y 442.29,Z 645.574,A -85,B 0,C 180,E1 22018.976,E2 22018.976} C_VEL
LIN {X 0,Y 442.298,Z 645.573,A -85,B 0,C 180,E1 22015.117,E2 22015.117} C_VEL
LIN {X 0,Y 442.333,Z 645.569,A -85,B 0,C 180,E1 22011.402,E2 22011.402} C_VEL
LIN {X 0,Y 442.383,Z 645.746,A -85,B 0,C 180,E1 22008.035,E2 22008.035} C_VEL
LIN {X 0,Y 450.876,Z 673.346,A -85,B 0,C 180,E1 22004.977,E2 22004.977} C_VEL
LIN {X 0,Y 456.151,Z 692.831,A -85,B 0,C 180,E1 22002.892,E2 22002.892} C_VEL
LIN {X 0,Y 454.195,Z 736.152,A -85,B 0,C 180,E1 21999.122,E2 21999.122} C_VEL
LIN {X 0,Y 452.284,Z 777.355,A -85,B 0,C 180,E1 21995.547,E2 21995.547} C_VEL
LIN {X 0,Y 450.415,Z 821.092,A -85,B 0,C 180,E1 21991.768,E2 21991.768} C_VEL
LIN {X 0,Y 449.614,Z 842.094,A -85,B 0,C 180,E1 21989.989,E2 21989.989} C_VEL
LIN {X 0,Y 446.634,Z 984.499,A -85,B 0,C 180,E1 21987.139,E2 21987.139} C_VEL
LIN {X 0,Y 446.389,Z 1000.927,A -85,B 0,C 180,E1 21986.611,E2 21986.611} C_VEL
LIN {X 0,Y 445.872,Z 1018.375,A -85,B 0,C 180,E1 21985.785,E2 21985.785} C_VEL
LIN {X 0,Y 445.275,Z 1033.808,A -85,B 0,C 180,E1 21984.789,E2 21984.789} C_VEL
LIN {X 0,Y 444.577,Z 1048.313,A -85,B 0,C 180,E1 21983.596,E2 21983.596} C_VEL
LIN {X 0,Y 443.791,Z 1062.62,A -85,B 0,C 180,E1 21982.099,E2 21982.099} C_VEL
LIN {X 0,Y 443.092,Z 1074.452,A -85,B 0,C 180,E1 21980.536,E2 21980.536} C_VEL
LIN {X 0,Y 442.502,Z 1084.766,A -85,B 0,C 180,E1 21978.849,E2 21978.849} C_VEL
LIN {X 0,Y 442.026,Z 1094.023,A -85,B 0,C 180,E1 21976.902,E2 21976.902} C_VEL
LIN {X 0,Y 441.748,Z 1100.658,A -85,B 0,C 180,E1 21975.085,E2 21975.085} C_VEL
LIN {X 0,Y 441.597,Z 1105.631,A -85,B 0,C 180,E1 21973.199,E2 21973.199} C_VEL
LIN {X 0,Y 441.613,Z 1109.047,A -85,B 0,C 180,E1 21971.358,E2 21971.358} C_VEL
LIN {X 0,Y 441.766,Z 1110.96,A -85,B 0,C 180,E1 21969.322,E2 21969.322} C_VEL
LIN {X 0,Y 442.1,Z 1111.078,A -85,B 0,C 180,E1 21967.273,E2 21967.273} C_VEL
LIN {X 0,Y 442.605,Z 1109.454,A -85,B 0,C 180,E1 21965.312,E2 21965.312} C_VEL
LIN {X 0,Y 443.361,Z 1105.805,A -85,B 0,C 180,E1 21963.229,E2 21963.229} C_VEL
LIN {X 0,Y 444.31,Z 1100.461,A -85,B 0,C 180,E1 21961.287,E2 21961.287} C_VEL
LIN {X 0,Y 445.508,Z 1093.064,A -85,B 0,C 180,E1 21959.354,E2 21959.354} C_VEL
LIN {X 0,Y 446.759,Z 1084.711,A -85,B 0,C 180,E1 21957.688,E2 21957.688} C_VEL
LIN {X 0,Y 448.195,Z 1074.183,A -85,B 0,C 180,E1 21956.032,E2 21956.032} C_VEL
LIN {X 0,Y 449.589,Z 1062.422,A -85,B 0,C 180,E1 21954.574,E2 21954.574} C_VEL
LIN {X 0,Y 450.931,Z 1049.014,A -85,B 0,C 180,E1 21953.248,E2 21953.248} C_VEL
LIN {X 0,Y 452.174,Z 1033.495,A -85,B 0,C 180,E1 21952.053,E2 21952.053} C_VEL
LIN {X 0,Y 453.093,Z 1018.328,A -85,B 0,C 180,E1 21951.175,E2 21951.175} C_VEL
LIN {X 0,Y 453.825,Z 1000.023,A -85,B 0,C 180,E1 21950.402,E2 21950.402} C_VEL
LIN {X 0,Y 454.124,Z 980.788,A -85,B 0,C 180,E1 21949.888,E2 21949.888} C_VEL
LIN {X 0,Y 458.411,Z 880.704,A -85,B 0,C 180,E1 21947.655,E2 21947.655} C_VEL
LIN {X 0,Y 459.829,Z 854.278,A -85,B 0,C 180,E1 21947.055,E2 21947.055} C_VEL
LIN {X 0,Y 460.449,Z 848.36,A -85,B 0,C 180,E1 21946.562,E2 21946.562} C_VEL
LIN {X 0,Y 463.285,Z 807.419,A -85,B 0,C 180,E1 21942.987,E2 21942.987} C_VEL
LIN {X 0,Y 466.318,Z 765.621,A -85,B 0,C 180,E1 21939.344,E2 21939.344} C_VEL
LIN {X 0,Y 469.883,Z 721.232,A -85,B 0,C 180,E1 21935.481,E2 21935.481} C_VEL
LIN {X 0,Y 470.998,Z 707.31,A -85,B 0,C 180,E1 21934.267,E2 21934.267} C_VEL
LIN {X 0,Y 467.929,Z 696.012,A -85,B 0,C 180,E1 21932.648,E2 21932.648} C_VEL
LIN {X 0,Y 464.116,Z 685.383,A -85,B 0,C 180,E1 21930.861,E2 21930.861} C_VEL
LIN {X 0,Y 459.949,Z 675.657,A -85,B 0,C 180,E1 21928.923,E2 21928.923} C_VEL
LIN {X 0,Y 457.277,Z 670.546,A -85,B 0,C 180,E1 21927.681,E2 21927.681} C_VEL
LIN {X 0,Y 455.454,Z 666.971,A -85,B 0,C 180,E1 21926.761,E2 21926.761} C_VEL
LIN {X 0,Y 453.419,Z 663.018,A -85,B 0,C 180,E1 21925.627,E2 21925.627} C_VEL
LIN {X 0,Y 450.696,Z 658.757,A -85,B 0,C 180,E1 21924.069,E2 21924.069} C_VEL
LIN {X 0,Y 450.202,Z 657.38,A -85,B 0,C 180,E1 21923.627,E2 21923.627} C_VEL
LIN {X 0,Y 447.535,Z 654.245,A -85,B 0,C 180,E1 21921.85,E2 21921.85} C_VEL
LIN {X 0,Y 446.705,Z 651.724,A -85,B 0,C 180,E1 21920.753,E2 21920.753} C_VEL
LIN {X 0,Y 444.266,Z 650.01,A -85,B 0,C 180,E1 21917.96,E2 21917.96} C_VEL
LIN {X 0,Y 444.006,Z 650.684,A -85,B 0,C 180,E1 21917.585,E2 21917.585} C_VEL
LIN {X 0,Y 450.815,Z 670.488,A -85,B 0,C 180,E1 21914.239,E2 21914.239} C_VEL
LIN {X 0,Y 452.123,Z 674.344,A -85,B 0,C 180,E1 21913.657,E2 21913.657} C_VEL
LIN {X 0,Y 469.612,Z 708.462,A -85,B 0,C 180,E1 21911.245,E2 21911.245} C_VEL
LIN {X 0,Y 478.435,Z 727.02,A -85,B 0,C 180,E1 21910.081,E2 21910.081} C_VEL
LIN {X 0,Y 480.452,Z 740.088,A -85,B 0,C 180,E1 21909.614,E2 21909.614} C_VEL
LIN {X 0,Y 468.214,Z 980.596,A -85,B 0,C 180,E1 21904.952,E2 21904.952} C_VEL
LIN {X 0,Y 466.27,Z 1004.302,A -85,B 0,C 180,E1 21904.271,E2 21904.271} C_VEL
LIN {X 0,Y 464.037,Z 1026.604,A -85,B 0,C 180,E1 21903.401,E2 21903.401} C_VEL
LIN {X 0,Y 461.517,Z 1048.258,A -85,B 0,C 180,E1 21902.331,E2 21902.331} C_VEL
LIN {X 0,Y 458.861,Z 1068.798,A -85,B 0,C 180,E1 21901.085,E2 21901.085} C_VEL
LIN {X 0,Y 456.076,Z 1088.778,A -85,B 0,C 180,E1 21899.626,E2 21899.626} C_VEL
LIN {X 0,Y 453.13,Z 1108.568,A -85,B 0,C 180,E1 21897.889,E2 21897.889} C_VEL
LIN {X 0,Y 450.468,Z 1126.089,A -85,B 0,C 180,E1 21896.069,E2 21896.069} C_VEL
LIN {X 0,Y 447.851,Z 1143.253,A -85,B 0,C 180,E1 21893.973,E2 21893.973} C_VEL
LIN {X 0,Y 445.696,Z 1158.008,A -85,B 0,C 180,E1 21891.862,E2 21891.862} C_VEL
LIN {X 0,Y 443.855,Z 1171.35,A -85,B 0,C 180,E1 21889.61,E2 21889.61} C_VEL
LIN {X 0,Y 442.377,Z 1183.339,A -85,B 0,C 180,E1 21887.221,E2 21887.221} C_VEL
LIN {X 0,Y 441.274,Z 1193.966,A -85,B 0,C 180,E1 21884.699,E2 21884.699} C_VEL
LIN {X 0,Y 440.583,Z 1202.677,A -85,B 0,C 180,E1 21882.182,E2 21882.182} C_VEL
LIN {X 0,Y 440.216,Z 1209.587,A -85,B 0,C 180,E1 21879.668,E2 21879.668} C_VEL
LIN {X 0,Y 440.083,Z 1215.159,A -85,B 0,C 180,E1 21877.045,E2 21877.045} C_VEL
LIN {X 0,Y 440.081,Z 1218.824,A -85,B 0,C 180,E1 21874.559,E2 21874.559} C_VEL
LIN {X 0,Y 440.123,Z 1221.166,A -85,B 0,C 180,E1 21871.821,E2 21871.821} C_VEL
LIN {X 0,Y 440.116,Z 1221.8,A -85,B 0,C 180,E1 21869.347,E2 21869.347} C_VEL
LIN {X 0,Y 440.068,Z 1220.807,A -85,B 0,C 180,E1 21866.742,E2 21866.742} C_VEL
LIN {X 0,Y 440.026,Z 1218.318,A -85,B 0,C 180,E1 21864.129,E2 21864.129} C_VEL
LIN {X 0,Y 440.096,Z 1214.368,A -85,B 0,C 180,E1 21861.638,E2 21861.638} C_VEL
LIN {X 0,Y 440.397,Z 1208.331,A -85,B 0,C 180,E1 21858.871,E2 21858.871} C_VEL
LIN {X 0,Y 441.048,Z 1200.839,A -85,B 0,C 180,E1 21856.227,E2 21856.227} C_VEL
LIN {X 0,Y 442.151,Z 1191.378,A -85,B 0,C 180,E1 21853.578,E2 21853.578} C_VEL
LIN {X 0,Y 443.812,Z 1179.942,A -85,B 0,C 180,E1 21850.931,E2 21850.931} C_VEL
LIN {X 0,Y 445.992,Z 1167.022,A -85,B 0,C 180,E1 21848.426,E2 21848.426} C_VEL
LIN {X 0,Y 448.706,Z 1152.324,A -85,B 0,C 180,E1 21846.017,E2 21846.017} C_VEL
LIN {X 0,Y 451.907,Z 1135.813,A -85,B 0,C 180,E1 21843.734,E2 21843.734} C_VEL
LIN {X 0,Y 455.391,Z 1118.45,A -85,B 0,C 180,E1 21841.687,E2 21841.687} C_VEL
LIN {X 0,Y 459.342,Z 1099.083,A -85,B 0,C 180,E1 21839.738,E2 21839.738} C_VEL
LIN {X 0,Y 463.449,Z 1078.797,A -85,B 0,C 180,E1 21838.008,E2 21838.008} C_VEL
LIN {X 0,Y 467.76,Z 1057.182,A -85,B 0,C 180,E1 21836.455,E2 21836.455} C_VEL
LIN {X 0,Y 472.286,Z 1033.661,A -85,B 0,C 180,E1 21835.061,E2 21835.061} C_VEL
LIN {X 0,Y 476.728,Z 1009.211,A -85,B 0,C 180,E1 21833.886,E2 21833.886} C_VEL
LIN {X 0,Y 481.046,Z 983.94,A -85,B 0,C 180,E1 21832.938,E2 21832.938} C_VEL
LIN {X 0,Y 485.116,Z 955.402,A -85,B 0,C 180,E1 21832.104,E2 21832.104} C_VEL
LIN {X 0,Y 494.443,Z 887.843,A -85,B 0,C 180,E1 21830.298,E2 21830.298} C_VEL
LIN {X 0,Y 506.617,Z 816.82,A -85,B 0,C 180,E1 21828.354,E2 21828.354} C_VEL
LIN {X 0,Y 520.247,Z 750.219,A -85,B 0,C 180,E1 21826.56,E2 21826.56} C_VEL
LIN {X 0,Y 520.08,Z 746.733,A -85,B 0,C 180,E1 21825.661,E2 21825.661} C_VEL
LIN {X 0,Y 520.176,Z 744.399,A -85,B 0,C 180,E1 21824.508,E2 21824.508} C_VEL
LIN {X 0,Y 520.523,Z 743.81,A -85,B 0,C 180,E1 21823.754,E2 21823.754} C_VEL
LIN {X 0,Y 521.202,Z 744.299,A -85,B 0,C 180,E1 21822.825,E2 21822.825} C_VEL
LIN {X 0,Y 505.989,Z 816.748,A -85,B 0,C 180,E1 21820.867,E2 21820.867} C_VEL
LIN {X 0,Y 494.171,Z 884.238,A -85,B 0,C 180,E1 21819.017,E2 21819.017} C_VEL
LIN {X 0,Y 484.483,Z 952.404,A -85,B 0,C 180,E1 21817.135,E2 21817.135} C_VEL
LIN {X 0,Y 480.991,Z 975.751,A -85,B 0,C 180,E1 21816.26,E2 21816.26} C_VEL
LIN {X 0,Y 477.197,Z 998.372,A -85,B 0,C 180,E1 21815.187,E2 21815.187} C_VEL
LIN {X 0,Y 472.999,Z 1021.148,A -85,B 0,C 180,E1 21813.852,E2 21813.852} C_VEL
LIN {X 0,Y 468.687,Z 1042.841,A -85,B 0,C 180,E1 21812.306,E2 21812.306} C_VEL
LIN {X 0,Y 464.346,Z 1063.364,A -85,B 0,C 180,E1 21810.545,E2 21810.545} C_VEL
LIN {X 0,Y 460.32,Z 1081.536,A -85,B 0,C 180,E1 21808.691,E2 21808.691} C_VEL
LIN {X 0,Y 456.619,Z 1097.736,A -85,B 0,C 180,E1 21806.746,E2 21806.746} C_VEL
LIN {X 0,Y 452.993,Z 1113.503,A -85,B 0,C 180,E1 21804.52,E2 21804.52} C_VEL
LIN {X 0,Y 449.824,Z 1127.375,A -85,B 0,C 180,E1 21802.205,E2 21802.205} C_VEL
LIN {X 0,Y 447.067,Z 1139.755,A -85,B 0,C 180,E1 21799.74,E2 21799.74} C_VEL
LIN {X 0,Y 444.867,Z 1150.06,A -85,B 0,C 180,E1 21797.261,E2 21797.261} C_VEL
LIN {X 0,Y 443.04,Z 1159.45,A -85,B 0,C 180,E1 21794.511,E2 21794.511} C_VEL
LIN {X 0,Y 441.807,Z 1166.614,A -85,B 0,C 180,E1 21791.888,E2 21791.888} C_VEL
LIN {X 0,Y 440.994,Z 1172.046,A -85,B 0,C 180,E1 21789.267,E2 21789.267} C_VEL
LIN {X 0,Y 440.496,Z 1176.07,A -85,B 0,C 180,E1 21786.52,E2 21786.52} C_VEL
LIN {X 0,Y 440.257,Z 1178.441,A -85,B 0,C 180,E1 21783.91,E2 21783.91} C_VEL
LIN {X 0,Y 440.153,Z 1179.217,A -85,B 0,C 180,E1 21781.304,E2 21781.304} C_VEL
LIN {X 0,Y 440.109,Z 1178.444,A -85,B 0,C 180,E1 21778.499,E2 21778.499} C_VEL
LIN {X 0,Y 440.14,Z 1176.123,A -85,B 0,C 180,E1 21775.8,E2 21775.8} C_VEL
LIN {X 0,Y 440.281,Z 1172.266,A -85,B 0,C 180,E1 21773.221,E2 21773.221} C_VEL
LIN {X 0,Y 440.618,Z 1166.5,A -85,B 0,C 180,E1 21770.468,E2 21770.468} C_VEL
LIN {X 0,Y 441.237,Z 1159.298,A -85,B 0,C 180,E1 21767.837,E2 21767.837} C_VEL
LIN {X 0,Y 442.2,Z 1150.148,A -85,B 0,C 180,E1 21765.199,E2 21765.199} C_VEL
LIN {X 0,Y 443.529,Z 1139.53,A -85,B 0,C 180,E1 21762.691,E2 21762.691} C_VEL
LIN {X 0,Y 445.317,Z 1126.833,A -85,B 0,C 180,E1 21760.185,E2 21760.185} C_VEL
LIN {X 0,Y 447.337,Z 1113.445,A -85,B 0,C 180,E1 21757.947,E2 21757.947} C_VEL
LIN {X 0,Y 449.705,Z 1098.126,A -85,B 0,C 180,E1 21755.785,E2 21755.785} C_VEL
LIN {X 0,Y 452.166,Z 1082.259,A -85,B 0,C 180,E1 21753.873,E2 21753.873} C_VEL
LIN {X 0,Y 454.91,Z 1064.241,A -85,B 0,C 180,E1 21752.017,E2 21752.017} C_VEL
LIN {X 0,Y 457.593,Z 1045.923,A -85,B 0,C 180,E1 21750.411,E2 21750.411} C_VEL
LIN {X 0,Y 460.254,Z 1025.995,A -85,B 0,C 180,E1 21748.95,E2 21748.95} C_VEL
LIN {X 0,Y 462.828,Z 1005.021,A -85,B 0,C 180,E1 21747.673,E2 21747.673} C_VEL
LIN {X 0,Y 465.25,Z 982.258,A -85,B 0,C 180,E1 21746.551,E2 21746.551} C_VEL
LIN {X 0,Y 467.236,Z 959.916,A -85,B 0,C 180,E1 21745.686,E2 21745.686} C_VEL
LIN {X 0,Y 468.904,Z 936.696,A -85,B 0,C 180,E1 21745.018,E2 21745.018} C_VEL
LIN {X 0,Y 480.122,Z 712.507,A -85,B 0,C 180,E1 21740.687,E2 21740.687} C_VEL
LIN {X 0,Y 460.859,Z 677.96,A -85,B 0,C 180,E1 21738.253,E2 21738.253} C_VEL
LIN {X 0,Y 444.017,Z 649.526,A -85,B 0,C 180,E1 21735.967,E2 21735.967} C_VEL
LIN {X 0,Y 442.448,Z 646.128,A -85,B 0,C 180,E1 21735.721,E2 21735.721} C_VEL
LIN {X 0,Y 442.356,Z 645.567,A -85,B 0,C 180,E1 21735.659,E2 21735.659} C_VEL
LIN {X 0,Y 442.351,Z 645.565,A -85,B 0,C 180,E1 21731.96,E2 21731.96} C_VEL
LIN {X 0,Y 442.339,Z 645.565,A -85,B 0,C 180,E1 21728.107,E2 21728.107} C_VEL
LIN {X 0,Y 442.358,Z 645.567,A -85,B 0,C 180,E1 21724.253,E2 21724.253} C_VEL
LIN {X 0,Y 442.356,Z 645.567,A -85,B 0,C 180,E1 21720.556,E2 21720.556} C_VEL
LIN {X 0,Y 442.339,Z 645.567,A -85,B 0,C 180,E1 21716.879,E2 21716.879} C_VEL
LIN {X 0,Y 442.314,Z 645.569,A -85,B 0,C 180,E1 21713.164,E2 21713.164} C_VEL
LIN {X 0,Y 442.332,Z 645.567,A -85,B 0,C 180,E1 21709.41,E2 21709.41} C_VEL
LIN {X 0,Y 442.366,Z 645.564,A -85,B 0,C 180,E1 21705.605,E2 21705.605} C_VEL
LIN {X 0,Y 442.35,Z 645.567,A -85,B 0,C 180,E1 21701.851,E2 21701.851} C_VEL
LIN {X 0,Y 442.32,Z 645.56,A -85,B 0,C 180,E1 21698.058,E2 21698.058} C_VEL
LIN {X 0,Y 442.291,Z 645.57,A -85,B 0,C 180,E1 21694.41,E2 21694.41} C_VEL
LIN {X 0,Y 442.315,Z 645.569,A -85,B 0,C 180,E1 21690.649,E2 21690.649} C_VEL
LIN {X 0,Y 442.355,Z 645.552,A -85,B 0,C 180,E1 21687.022,E2 21687.022} C_VEL
LIN {X 0,Y 442.347,Z 645.565,A -85,B 0,C 180,E1 21683.252,E2 21683.252} C_VEL
LIN {X 0,Y 442.314,Z 645.552,A -85,B 0,C 180,E1 21679.51,E2 21679.51} C_VEL
LIN {X 0,Y 442.282,Z 645.572,A -85,B 0,C 180,E1 21675.736,E2 21675.736} C_VEL
LIN {X 0,Y 442.29,Z 645.57,A -85,B 0,C 180,E1 21673.715,E2 21673.715} C_VEL
LIN {X 0,Y 441.3,Z 645.696,A -85,B 0,C 180,E1 21672.717,E2 21672.717} C_VEL
LIN {X 0,Y 434.815,Z 646.502,A -85,B 0,C 180,E1 21669.832,E2 21669.832} C_VEL
LIN {X 0,Y 434.412,Z 646.554,A -85,B 0,C 180,E1 21669.171,E2 21669.171} C_VEL
LIN {X 0,Y 434.415,Z 646.559,A -85,B 0,C 180,E1 21665.381,E2 21665.381} C_VEL
LIN {X 0,Y 434.409,Z 646.557,A -85,B 0,C 180,E1 21661.698,E2 21661.698} C_VEL
LIN {X 0,Y 434.393,Z 646.56,A -85,B 0,C 180,E1 21658.037,E2 21658.037} C_VEL
LIN {X 0,Y 434.409,Z 646.559,A -85,B 0,C 180,E1 21654.11,E2 21654.11} C_VEL
LIN {X 0,Y 434.426,Z 646.554,A -85,B 0,C 180,E1 21650.394,E2 21650.394} C_VEL
LIN {X 0,Y 434.429,Z 646.648,A -85,B 0,C 180,E1 21648.484,E2 21648.484} C_VEL
LIN {X 0,Y 443.229,Z 675.112,A -85,B 0,C 180,E1 21645.28,E2 21645.28} C_VEL
LIN {X 0,Y 448.631,Z 695.039,A -85,B 0,C 180,E1 21643.133,E2 21643.133} C_VEL
LIN {X 0,Y 446.618,Z 737.489,A -85,B 0,C 180,E1 21639.401,E2 21639.401} C_VEL
LIN {X 0,Y 444.595,Z 779.475,A -85,B 0,C 180,E1 21635.724,E2 21635.724} C_VEL
LIN {X 0,Y 442.61,Z 823.786,A -85,B 0,C 180,E1 21631.857,E2 21631.857} C_VEL
LIN {X 0,Y 441.898,Z 842.946,A -85,B 0,C 180,E1 21630.238,E2 21630.238} C_VEL
LIN {X 0,Y 438.774,Z 984.797,A -85,B 0,C 180,E1 21627.328,E2 21627.328} C_VEL
LIN {X 0,Y 438.526,Z 1001.276,A -85,B 0,C 180,E1 21626.797,E2 21626.797} C_VEL
LIN {X 0,Y 437.992,Z 1018.928,A -85,B 0,C 180,E1 21625.952,E2 21625.952} C_VEL
LIN {X 0,Y 437.381,Z 1034.394,A -85,B 0,C 180,E1 21624.943,E2 21624.943} C_VEL
LIN {X 0,Y 436.685,Z 1048.643,A -85,B 0,C 180,E1 21623.762,E2 21623.762} C_VEL
LIN {X 0,Y 435.917,Z 1062.293,A -85,B 0,C 180,E1 21622.328,E2 21622.328} C_VEL
LIN {X 0,Y 435.249,Z 1073.644,A -85,B 0,C 180,E1 21620.856,E2 21620.856} C_VEL
LIN {X 0,Y 434.592,Z 1084.681,A -85,B 0,C 180,E1 21619.066,E2 21619.066} C_VEL
LIN {X 0,Y 434.133,Z 1093.381,A -85,B 0,C 180,E1 21617.281,E2 21617.281} C_VEL
LIN {X 0,Y 433.801,Z 1101.082,A -85,B 0,C 180,E1 21615.231,E2 21615.231} C_VEL
LIN {X 0,Y 433.644,Z 1106.226,A -85,B 0,C 180,E1 21613.328,E2 21613.328} C_VEL
LIN {X 0,Y 433.659,Z 1109.979,A -85,B 0,C 180,E1 21611.299,E2 21611.299} C_VEL
LIN {X 0,Y 433.827,Z 1111.935,A -85,B 0,C 180,E1 21609.281,E2 21609.281} C_VEL
LIN {X 0,Y 434.2,Z 1112.123,A -85,B 0,C 180,E1 21607.14,E2 21607.14} C_VEL
LIN {X 0,Y 434.746,Z 1110.548,A -85,B 0,C 180,E1 21605.143,E2 21605.143} C_VEL
LIN {X 0,Y 435.561,Z 1106.927,A -85,B 0,C 180,E1 21603.024,E2 21603.024} C_VEL
LIN {X 0,Y 436.584,Z 1101.645,A -85,B 0,C 180,E1 21601.047,E2 21601.047} C_VEL
LIN {X 0,Y 437.87,Z 1094.322,A -85,B 0,C 180,E1 21599.081,E2 21599.081} C_VEL
LIN {X 0,Y 439.201,Z 1086.006,A -85,B 0,C 180,E1 21597.388,E2 21597.388} C_VEL
LIN {X 0,Y 440.717,Z 1075.493,A -85,B 0,C 180,E1 21595.704,E2 21595.704} C_VEL
LIN {X 0,Y 442.197,Z 1063.797,A -85,B 0,C 180,E1 21594.222,E2 21594.222} C_VEL
LIN {X 0,Y 443.639,Z 1050.572,A -85,B 0,C 180,E1 21592.877,E2 21592.877} C_VEL
LIN {X 0,Y 444.887,Z 1036.107,A -85,B 0,C 180,E1 21591.727,E2 21591.727} C_VEL
LIN {X 0,Y 445.714,Z 1023.719,A -85,B 0,C 180,E1 21590.963,E2 21590.963} C_VEL
LIN {X 0,Y 446.368,Z 1011.126,A -85,B 0,C 180,E1 21590.342,E2 21590.342} C_VEL
LIN {X 0,Y 446.863,Z 996.392,A -85,B 0,C 180,E1 21589.791,E2 21589.791} C_VEL
LIN {X 0,Y 447.916,Z 957.874,A -85,B 0,C 180,E1 21588.864,E2 21588.864} C_VEL
LIN {X 0,Y 453.21,Z 855.625,A -85,B 0,C 180,E1 21586.505,E2 21586.505} C_VEL
LIN {X 0,Y 454.074,Z 846.474,A -85,B 0,C 180,E1 21585.719,E2 21585.719} C_VEL
LIN {X 0,Y 457.434,Z 801.202,A -85,B 0,C 180,E1 21581.717,E2 21581.717} C_VEL
LIN {X 0,Y 460.855,Z 759.09,A -85,B 0,C 180,E1 21578.019,E2 21578.019} C_VEL
LIN {X 0,Y 464.987,Z 713.281,A -85,B 0,C 180,E1 21573.978,E2 21573.978} C_VEL
LIN {X 0,Y 464.979,Z 710.575,A -85,B 0,C 180,E1 21573.703,E2 21573.703} C_VEL
LIN {X 0,Y 461.584,Z 698.242,A -85,B 0,C 180,E1 21571.818,E2 21571.818} C_VEL
LIN {X 0,Y 457.974,Z 688.216,A -85,B 0,C 180,E1 21569.999,E2 21569.999} C_VEL
LIN {X 0,Y 453.659,Z 678.214,A -85,B 0,C 180,E1 21567.813,E2 21567.813} C_VEL
LIN {X 0,Y 451.066,Z 673.321,A -85,B 0,C 180,E1 21566.454,E2 21566.454} C_VEL
LIN {X 0,Y 449.079,Z 669.245,A -85,B 0,C 180,E1 21565.24,E2 21565.24} C_VEL
LIN {X 0,Y 446.9,Z 665.652,A -85,B 0,C 180,E1 21563.867,E2 21563.867} C_VEL
LIN {X 0,Y 446.221,Z 664.21,A -85,B 0,C 180,E1 21563.337,E2 21563.337} C_VEL
LIN {X 0,Y 443.91,Z 661.04,A -85,B 0,C 180,E1 21561.559,E2 21561.559} C_VEL
LIN {X 0,Y 443.384,Z 658.994,A -85,B 0,C 180,E1 21560.666,E2 21560.666} C_VEL
LIN {X 0,Y 441.206,Z 657.569,A -85,B 0,C 180,E1 21558.013,E2 21558.013} C_VEL
LIN {X 0,Y 439.589,Z 660.634,A -85,B 0,C 180,E1 21556.895,E2 21556.895} C_VEL
LIN {X 0,Y 439.442,Z 661.337,A -85,B 0,C 180,E1 21556.535,E2 21556.535} C_VEL
LIN {X 0,Y 443.761,Z 673.976,A -85,B 0,C 180,E1 21554.437,E2 21554.437} C_VEL
LIN {X 0,Y 461.507,Z 708.451,A -85,B 0,C 180,E1 21551.929,E2 21551.929} C_VEL
LIN {X 0,Y 472.042,Z 730.504,A -85,B 0,C 180,E1 21550.506,E2 21550.506} C_VEL
LIN {X 0,Y 473.661,Z 741.476,A -85,B 0,C 180,E1 21550.111,E2 21550.111} C_VEL
LIN {X 0,Y 461.001,Z 980.455,A -85,B 0,C 180,E1 21545.38,E2 21545.38} C_VEL
LIN {X 0,Y 458.985,Z 1004.311,A -85,B 0,C 180,E1 21544.682,E2 21544.682} C_VEL
LIN {X 0,Y 456.663,Z 1026.784,A -85,B 0,C 180,E1 21543.787,E2 21543.787} C_VEL
LIN {X 0,Y 454.134,Z 1047.89,A -85,B 0,C 180,E1 21542.725,E2 21542.725} C_VEL
LIN {X 0,Y 451.366,Z 1068.677,A -85,B 0,C 180,E1 21541.443,E2 21541.443} C_VEL
LIN {X 0,Y 448.495,Z 1088.69,A -85,B 0,C 180,E1 21539.957,E2 21539.957} C_VEL
LIN {X 0,Y 445.471,Z 1108.447,A -85,B 0,C 180,E1 21538.193,E2 21538.193} C_VEL
LIN {X 0,Y 442.734,Z 1125.936,A -85,B 0,C 180,E1 21536.343,E2 21536.343} C_VEL
LIN {X 0,Y 440.044,Z 1143.091,A -85,B 0,C 180,E1 21534.211,E2 21534.211} C_VEL
LIN {X 0,Y 437.893,Z 1157.429,A -85,B 0,C 180,E1 21532.131,E2 21532.131} C_VEL
LIN {X 0,Y 435.988,Z 1170.814,A -85,B 0,C 180,E1 21529.839,E2 21529.839} C_VEL
LIN {X 0,Y 434.456,Z 1182.855,A -85,B 0,C 180,E1 21527.407,E2 21527.407} C_VEL
LIN {X 0,Y 433.314,Z 1193.522,A -85,B 0,C 180,E1 21524.839,E2 21524.839} C_VEL
LIN {X 0,Y 432.601,Z 1202.253,A -85,B 0,C 180,E1 21522.275,E2 21522.275} C_VEL
LIN {X 0,Y 432.225,Z 1209.164,A -85,B 0,C 180,E1 21519.72,E2 21519.72} C_VEL
LIN {X 0,Y 432.093,Z 1214.758,A -85,B 0,C 180,E1 21517.043,E2 21517.043} C_VEL
LIN {X 0,Y 432.095,Z 1218.419,A -85,B 0,C 180,E1 21514.511,E2 21514.511} C_VEL
LIN {X 0,Y 432.136,Z 1220.685,A -85,B 0,C 180,E1 21511.854,E2 21511.854} C_VEL
LIN {X 0,Y 432.129,Z 1221.343,A -85,B 0,C 180,E1 21509.468,E2 21509.468} C_VEL
LIN {X 0,Y 432.075,Z 1220.523,A -85,B 0,C 180,E1 21506.814,E2 21506.814} C_VEL
LIN {X 0,Y 432.028,Z 1218.3,A -85,B 0,C 180,E1 21504.287,E2 21504.287} C_VEL
LIN {X 0,Y 432.098,Z 1214.329,A -85,B 0,C 180,E1 21501.616,E2 21501.616} C_VEL
LIN {X 0,Y 432.388,Z 1208.801,A -85,B 0,C 180,E1 21498.933,E2 21498.933} C_VEL
LIN {X 0,Y 433.047,Z 1201.46,A -85,B 0,C 180,E1 21496.24,E2 21496.24} C_VEL
LIN {X 0,Y 434.254,Z 1191.801,A -85,B 0,C 180,E1 21493.409,E2 21493.409} C_VEL
LIN {X 0,Y 436.001,Z 1180.592,A -85,B 0,C 180,E1 21490.715,E2 21490.715} C_VEL
LIN {X 0,Y 438.291,Z 1167.93,A -85,B 0,C 180,E1 21488.168,E2 21488.168} C_VEL
LIN {X 0,Y 441.054,Z 1153.757,A -85,B 0,C 180,E1 21485.773,E2 21485.773} C_VEL
LIN {X 0,Y 444.476,Z 1137.296,A -85,B 0,C 180,E1 21483.404,E2 21483.404} C_VEL
LIN {X 0,Y 448.364,Z 1119.26,A -85,B 0,C 180,E1 21481.202,E2 21481.202} C_VEL
LIN {X 0,Y 452.525,Z 1100.292,A -85,B 0,C 180,E1 21479.234,E2 21479.234} C_VEL
LIN {X 0,Y 456.987,Z 1079.869,A -85,B 0,C 180,E1 21477.434,E2 21477.434} C_VEL
LIN {X 0,Y 461.9,Z 1056.925,A -85,B 0,C 180,E1 21475.747,E2 21475.747} C_VEL
LIN {X 0,Y 466.886,Z 1032.902,A -85,B 0,C 180,E1 21474.295,E2 21474.295} C_VEL
LIN {X 0,Y 471.854,Z 1007.883,A -85,B 0,C 180,E1 21473.075,E2 21473.075} C_VEL
LIN {X 0,Y 476.581,Z 982.328,A -85,B 0,C 180,E1 21472.105,E2 21472.105} C_VEL
LIN {X 0,Y 481.17,Z 952.668,A -85,B 0,C 180,E1 21471.223,E2 21471.223} C_VEL
LIN {X 0,Y 491.479,Z 885.609,A -85,B 0,C 180,E1 21469.38,E2 21469.38} C_VEL
LIN {X 0,Y 504.859,Z 814.729,A -85,B 0,C 180,E1 21467.411,E2 21467.411} C_VEL
LIN {X 0,Y 517.94,Z 755.47,A -85,B 0,C 180,E1 21465.798,E2 21465.798} C_VEL
LIN {X 0,Y 518.012,Z 753.241,A -85,B 0,C 180,E1 21465.051,E2 21465.051} C_VEL
LIN {X 0,Y 518.478,Z 751.556,A -85,B 0,C 180,E1 21463.84,E2 21463.84} C_VEL
LIN {X 0,Y 518.597,Z 751.805,A -85,B 0,C 180,E1 21463.521,E2 21463.521} C_VEL
LIN {X 0,Y 501.933,Z 826.359,A -85,B 0,C 180,E1 21461.492,E2 21461.492} C_VEL
LIN {X 0,Y 489.327,Z 893.77,A -85,B 0,C 180,E1 21459.616,E2 21459.616} C_VEL
LIN {X 0,Y 480.055,Z 953.613,A -85,B 0,C 180,E1 21457.914,E2 21457.914} C_VEL
LIN {X 0,Y 476.105,Z 977.385,A -85,B 0,C 180,E1 21456.993,E2 21456.993} C_VEL
LIN {X 0,Y 471.871,Z 1000.361,A -85,B 0,C 180,E1 21455.869,E2 21455.869} C_VEL
LIN {X 0,Y 467.428,Z 1022.502,A -85,B 0,C 180,E1 21454.535,E2 21454.535} C_VEL
LIN {X 0,Y 462.682,Z 1044.489,A -85,B 0,C 180,E1 21452.925,E2 21452.925} C_VEL
LIN {X 0,Y 457.947,Z 1065.286,A -85,B 0,C 180,E1 21451.092,E2 21451.092} C_VEL
LIN {X 0,Y 453.444,Z 1084.257,A -85,B 0,C 180,E1 21449.095,E2 21449.095} C_VEL
LIN {X 0,Y 449.322,Z 1100.98,A -85,B 0,C 180,E1 21447.001,E2 21447.001} C_VEL
LIN {X 0,Y 445.642,Z 1115.833,A -85,B 0,C 180,E1 21444.81,E2 21444.81} C_VEL
LIN {X 0,Y 442.151,Z 1130.025,A -85,B 0,C 180,E1 21442.331,E2 21442.331} C_VEL
LIN {X 0,Y 439.295,Z 1142.026,A -85,B 0,C 180,E1 21439.827,E2 21439.827} C_VEL
LIN {X 0,Y 436.923,Z 1152.582,A -85,B 0,C 180,E1 21437.173,E2 21437.173} C_VEL
LIN {X 0,Y 435.128,Z 1161.122,A -85,B 0,C 180,E1 21434.508,E2 21434.508} C_VEL
LIN {X 0,Y 433.801,Z 1168.255,A -85,B 0,C 180,E1 21431.705,E2 21431.705} C_VEL
LIN {X 0,Y 432.996,Z 1173.438,A -85,B 0,C 180,E1 21429.037,E2 21429.037} C_VEL
LIN {X 0,Y 432.494,Z 1177.123,A -85,B 0,C 180,E1 21426.241,E2 21426.241} C_VEL
LIN {X 0,Y 432.252,Z 1179.172,A -85,B 0,C 180,E1 21423.451,E2 21423.451} C_VEL
LIN {X 0,Y 432.154,Z 1179.686,A -85,B 0,C 180,E1 21420.798,E2 21420.798} C_VEL
LIN {X 0,Y 432.116,Z 1178.588,A -85,B 0,C 180,E1 21418.146,E2 21418.146} C_VEL
LIN {X 0,Y 432.163,Z 1175.879,A -85,B 0,C 180,E1 21415.358,E2 21415.358} C_VEL
LIN {X 0,Y 432.344,Z 1171.758,A -85,B 0,C 180,E1 21412.695,E2 21412.695} C_VEL
LIN {X 0,Y 432.722,Z 1165.893,A -85,B 0,C 180,E1 21410.023,E2 21410.023} C_VEL
LIN {X 0,Y 433.438,Z 1157.906,A -85,B 0,C 180,E1 21407.208,E2 21407.208} C_VEL
LIN {X 0,Y 434.462,Z 1148.884,A -85,B 0,C 180,E1 21404.648,E2 21404.648} C_VEL
LIN {X 0,Y 435.904,Z 1137.95,A -85,B 0,C 180,E1 21402.102,E2 21402.102} C_VEL
LIN {X 0,Y 437.714,Z 1125.536,A -85,B 0,C 180,E1 21399.686,E2 21399.686} C_VEL
LIN {X 0,Y 439.984,Z 1110.883,A -85,B 0,C 180,E1 21397.277,E2 21397.277} C_VEL
LIN {X 0,Y 442.439,Z 1095.636,A -85,B 0,C 180,E1 21395.147,E2 21395.147} C_VEL
LIN {X 0,Y 445.097,Z 1078.923,A -85,B 0,C 180,E1 21393.161,E2 21393.161} C_VEL
LIN {X 0,Y 447.823,Z 1061.329,A -85,B 0,C 180,E1 21391.388,E2 21391.388} C_VEL
LIN {X 0,Y 450.728,Z 1041.511,A -85,B 0,C 180,E1 21389.694,E2 21389.694} C_VEL
LIN {X 0,Y 453.437,Z 1021.729,A -85,B 0,C 180,E1 21388.273,E2 21388.273} C_VEL
LIN {X 0,Y 456.09,Z 1000.162,A -85,B 0,C 180,E1 21386.994,E2 21386.994} C_VEL
LIN {X 0,Y 458.404,Z 978.125,A -85,B 0,C 180,E1 21385.95,E2 21385.95} C_VEL
LIN {X 0,Y 460.364,Z 955.737,A -85,B 0,C 180,E1 21385.121,E2 21385.121} C_VEL
LIN {X 0,Y 461.997,Z 931.47,A -85,B 0,C 180,E1 21384.464,E2 21384.464} C_VEL
LIN {X 0,Y 473.286,Z 715.288,A -85,B 0,C 180,E1 21380.219,E2 21380.219} C_VEL
LIN {X 0,Y 454.445,Z 681.536,A -85,B 0,C 180,E1 21377.789,E2 21377.789} C_VEL
LIN {X 0,Y 438.201,Z 654.088,A -85,B 0,C 180,E1 21375.533,E2 21375.533} C_VEL
LIN {X 0,Y 436.189,Z 650.688,A -85,B 0,C 180,E1 21375.241,E2 21375.241} C_VEL
LIN {X 0,Y 434.525,Z 647.317,A -85,B 0,C 180,E1 21374.983,E2 21374.983} C_VEL
LIN {X 0,Y 434.393,Z 646.556,A -85,B 0,C 180,E1 21374.91,E2 21374.91} C_VEL
LIN {X 0,Y 434.357,Z 646.564,A -85,B 0,C 180,E1 21371.176,E2 21371.176} C_VEL
LIN {X 0,Y 434.362,Z 646.559,A -85,B 0,C 180,E1 21367.426,E2 21367.426} C_VEL
LIN {X 0,Y 434.405,Z 646.556,A -85,B 0,C 180,E1 21363.693,E2 21363.693} C_VEL
LIN {X 0,Y 434.426,Z 646.551,A -85,B 0,C 180,E1 21359.965,E2 21359.965} C_VEL
LIN {X 0,Y 434.391,Z 646.553,A -85,B 0,C 180,E1 21356.23,E2 21356.23} C_VEL
LIN {X 0,Y 434.346,Z 646.557,A -85,B 0,C 180,E1 21352.468,E2 21352.468} C_VEL
LIN {X 0,Y 434.363,Z 646.556,A -85,B 0,C 180,E1 21348.663,E2 21348.663} C_VEL
LIN {X 0,Y 434.395,Z 646.555,A -85,B 0,C 180,E1 21344.831,E2 21344.831} C_VEL
LIN {X 0,Y 434.419,Z 646.555,A -85,B 0,C 180,E1 21341.015,E2 21341.015} C_VEL
LIN {X 0,Y 434.407,Z 646.548,A -85,B 0,C 180,E1 21337.263,E2 21337.263} C_VEL
LIN {X 0,Y 434.356,Z 646.555,A -85,B 0,C 180,E1 21333.565,E2 21333.565} C_VEL
LIN {X 0,Y 434.374,Z 646.559,A -85,B 0,C 180,E1 21329.87,E2 21329.87} C_VEL
LIN {X 0,Y 434.399,Z 646.539,A -85,B 0,C 180,E1 21326.174,E2 21326.174} C_VEL
LIN {X 0,Y 434.423,Z 646.555,A -85,B 0,C 180,E1 21322.33,E2 21322.33} C_VEL
LIN {X 0,Y 434.407,Z 646.534,A -85,B 0,C 180,E1 21318.585,E2 21318.585} C_VEL
LIN {X 0,Y 434.382,Z 646.561,A -85,B 0,C 180,E1 21314.789,E2 21314.789} C_VEL
LIN {X 0,Y 434.402,Z 646.559,A -85,B 0,C 180,E1 21311.064,E2 21311.064} C_VEL
LIN {X 0,Y 434.412,Z 646.554,A -85,B 0,C 180,E1 21309.171,E2 21309.171} C_VEL
LIN {X 0,Y 433.457,Z 646.677,A -85,B 0,C 180,E1 21308.155,E2 21308.155} C_VEL
LIN {X 0,Y 426.897,Z 647.493,A -85,B 0,C 180,E1 21305.22,E2 21305.22} C_VEL
LIN {X 0,Y 426.473,Z 647.542,A -85,B 0,C 180,E1 21304.546,E2 21304.546} C_VEL
LIN {X 0,Y 426.436,Z 647.549,A -85,B 0,C 180,E1 21300.812,E2 21300.812} C_VEL
LIN {X 0,Y 426.408,Z 647.553,A -85,B 0,C 180,E1 21297.045,E2 21297.045} C_VEL
LIN {X 0,Y 426.442,Z 647.548,A -85,B 0,C 180,E1 21293.115,E2 21293.115} C_VEL
LIN {X 0,Y 426.474,Z 647.544,A -85,B 0,C 180,E1 21289.22,E2 21289.22} C_VEL
LIN {X 0,Y 426.512,Z 647.764,A -85,B 0,C 180,E1 21288.932,E2 21288.932} C_VEL
LIN {X 0,Y 434.929,Z 674.818,A -85,B 0,C 180,E1 21285.825,E2 21285.825} C_VEL
LIN {X 0,Y 441.118,Z 697.293,A -85,B 0,C 180,E1 21283.373,E2 21283.373} C_VEL
LIN {X 0,Y 439.014,Z 739.654,A -85,B 0,C 180,E1 21279.618,E2 21279.618} C_VEL
LIN {X 0,Y 436.916,Z 781.815,A -85,B 0,C 180,E1 21275.895,E2 21275.895} C_VEL
LIN {X 0,Y 434.804,Z 826.841,A -85,B 0,C 180,E1 21271.928,E2 21271.928} C_VEL
LIN {X 0,Y 434.173,Z 843.716,A -85,B 0,C 180,E1 21270.492,E2 21270.492} C_VEL
LIN {X 0,Y 430.918,Z 985.113,A -85,B 0,C 180,E1 21267.524,E2 21267.524} C_VEL
LIN {X 0,Y 430.663,Z 1001.772,A -85,B 0,C 180,E1 21266.983,E2 21266.983} C_VEL
LIN {X 0,Y 430.166,Z 1018.029,A -85,B 0,C 180,E1 21266.205,E2 21266.205} C_VEL
LIN {X 0,Y 429.556,Z 1033.586,A -85,B 0,C 180,E1 21265.209,E2 21265.209} C_VEL
LIN {X 0,Y 428.793,Z 1048.989,A -85,B 0,C 180,E1 21263.929,E2 21263.929} C_VEL
LIN {X 0,Y 428.031,Z 1062.328,A -85,B 0,C 180,E1 21262.523,E2 21262.523} C_VEL
LIN {X 0,Y 427.318,Z 1074.196,A -85,B 0,C 180,E1 21260.974,E2 21260.974} C_VEL
LIN {X 0,Y 426.641,Z 1085.306,A -85,B 0,C 180,E1 21259.15,E2 21259.15} C_VEL
LIN {X 0,Y 426.172,Z 1094.098,A -85,B 0,C 180,E1 21257.332,E2 21257.332} C_VEL
LIN {X 0,Y 425.833,Z 1101.858,A -85,B 0,C 180,E1 21255.244,E2 21255.244} C_VEL
LIN {X 0,Y 425.681,Z 1107.1,A -85,B 0,C 180,E1 21253.305,E2 21253.305} C_VEL
LIN {X 0,Y 425.705,Z 1110.908,A -85,B 0,C 180,E1 21251.239,E2 21251.239} C_VEL
LIN {X 0,Y 425.896,Z 1112.933,A -85,B 0,C 180,E1 21249.183,E2 21249.183} C_VEL
LIN {X 0,Y 426.302,Z 1113.169,A -85,B 0,C 180,E1 21247.002,E2 21247.002} C_VEL
LIN {X 0,Y 426.893,Z 1111.653,A -85,B 0,C 180,E1 21244.969,E2 21244.969} C_VEL
LIN {X 0,Y 427.775,Z 1108.098,A -85,B 0,C 180,E1 21242.811,E2 21242.811} C_VEL
LIN {X 0,Y 428.795,Z 1103.303,A -85,B 0,C 180,E1 21240.932,E2 21240.932} C_VEL
LIN {X 0,Y 430.14,Z 1096.124,A -85,B 0,C 180,E1 21238.932,E2 21238.932} C_VEL
LIN {X 0,Y 431.543,Z 1088.029,A -85,B 0,C 180,E1 21237.208,E2 21237.208} C_VEL
LIN {X 0,Y 433.142,Z 1077.779,A -85,B 0,C 180,E1 21235.496,E2 21235.496} C_VEL
LIN {X 0,Y 434.718,Z 1066.473,A -85,B 0,C 180,E1 21233.99,E2 21233.99} C_VEL
LIN {X 0,Y 436.3,Z 1052.865,A -85,B 0,C 180,E1 21232.558,E2 21232.558} C_VEL
LIN {X 0,Y 437.545,Z 1039.614,A -85,B 0,C 180,E1 21231.455,E2 21231.455} C_VEL
LIN {X 0,Y 438.58,Z 1025.675,A -85,B 0,C 180,E1 21230.55,E2 21230.55} C_VEL
LIN {X 0,Y 439.337,Z 1012.564,A -85,B 0,C 180,E1 21229.88,E2 21229.88} C_VEL
LIN {X 0,Y 439.9,Z 997.836,A -85,B 0,C 180,E1 21229.309,E2 21229.309} C_VEL
LIN {X 0,Y 441.038,Z 959.258,A -85,B 0,C 180,E1 21228.353,E2 21228.353} C_VEL
LIN {X 0,Y 446.632,Z 856.963,A -85,B 0,C 180,E1 21225.94,E2 21225.94} C_VEL
LIN {X 0,Y 448.37,Z 837.41,A -85,B 0,C 180,E1 21224.21,E2 21224.21} C_VEL
LIN {X 0,Y 451.882,Z 794.162,A -85,B 0,C 180,E1 21220.344,E2 21220.344} C_VEL
LIN {X 0,Y 455.814,Z 750.735,A -85,B 0,C 180,E1 21216.467,E2 21216.467} C_VEL
LIN {X 0,Y 459.409,Z 715.252,A -85,B 0,C 180,E1 21213.29,E2 21213.29} C_VEL
LIN {X 0,Y 456.345,Z 703.586,A -85,B 0,C 180,E1 21211.465,E2 21211.465} C_VEL
LIN {X 0,Y 452.936,Z 693.751,A -85,B 0,C 180,E1 21209.631,E2 21209.631} C_VEL
LIN {X 0,Y 449.183,Z 684.493,A -85,B 0,C 180,E1 21207.524,E2 21207.524} C_VEL
LIN {X 0,Y 446.684,Z 679.615,A -85,B 0,C 180,E1 21206.123,E2 21206.123} C_VEL
LIN {X 0,Y 444.797,Z 675.663,A -85,B 0,C 180,E1 21204.864,E2 21204.864} C_VEL
LIN {X 0,Y 442.878,Z 671.751,A -85,B 0,C 180,E1 21203.411,E2 21203.411} C_VEL
LIN {X 0,Y 440.465,Z 668.059,A -85,B 0,C 180,E1 21201.34,E2 21201.34} C_VEL
LIN {X 0,Y 439.857,Z 666.146,A -85,B 0,C 180,E1 21200.406,E2 21200.406} C_VEL
LIN {X 0,Y 438.245,Z 665.089,A -85,B 0,C 180,E1 21198.221,E2 21198.221} C_VEL
LIN {X 0,Y 436.697,Z 667.913,A -85,B 0,C 180,E1 21197.109,E2 21197.109} C_VEL
LIN {X 0,Y 435.086,Z 672.22,A -85,B 0,C 180,E1 21195.617,E2 21195.617} C_VEL
LIN {X 0,Y 435.119,Z 673.01,A -85,B 0,C 180,E1 21195.315,E2 21195.315} C_VEL
LIN {X 0,Y 452.161,Z 705.999,A -85,B 0,C 180,E1 21192.807,E2 21192.807} C_VEL
LIN {X 0,Y 465.6,Z 733.676,A -85,B 0,C 180,E1 21190.949,E2 21190.949} C_VEL
LIN {X 0,Y 466.882,Z 742.813,A -85,B 0,C 180,E1 21190.618,E2 21190.618} C_VEL
LIN {X 0,Y 453.811,Z 980.104,A -85,B 0,C 180,E1 21185.822,E2 21185.822} C_VEL
LIN {X 0,Y 451.727,Z 1004.054,A -85,B 0,C 180,E1 21185.108,E2 21185.108} C_VEL
LIN {X 0,Y 449.304,Z 1026.8,A -85,B 0,C 180,E1 21184.186,E2 21184.186} C_VEL
LIN {X 0,Y 446.699,Z 1047.913,A -85,B 0,C 180,E1 21183.102,E2 21183.102} C_VEL
LIN {X 0,Y 443.738,Z 1069.447,A -85,B 0,C 180,E1 21181.743,E2 21181.743} C_VEL
LIN {X 0,Y 440.806,Z 1089.285,A -85,B 0,C 180,E1 21180.234,E2 21180.234} C_VEL
LIN {X 0,Y 437.824,Z 1108.268,A -85,B 0,C 180,E1 21178.507,E2 21178.507} C_VEL
LIN {X 0,Y 435.009,Z 1125.75,A -85,B 0,C 180,E1 21176.627,E2 21176.627} C_VEL
LIN {X 0,Y 432.244,Z 1142.903,A -85,B 0,C 180,E1 21174.458,E2 21174.458} C_VEL
LIN {X 0,Y 429.93,Z 1157.892,A -85,B 0,C 180,E1 21172.232,E2 21172.232} C_VEL
LIN {X 0,Y 427.923,Z 1171.747,A -85,B 0,C 180,E1 21169.802,E2 21169.802} C_VEL
LIN {X 0,Y 426.393,Z 1183.569,A -85,B 0,C 180,E1 21167.324,E2 21167.324} C_VEL
LIN {X 0,Y 425.263,Z 1194.031,A -85,B 0,C 180,E1 21164.708,E2 21164.708} C_VEL
LIN {X 0,Y 424.565,Z 1202.646,A -85,B 0,C 180,E1 21162.097,E2 21162.097} C_VEL
LIN {X 0,Y 424.213,Z 1209.382,A -85,B 0,C 180,E1 21159.495,E2 21159.495} C_VEL
LIN {X 0,Y 424.095,Z 1214.776,A -85,B 0,C 180,E1 21156.768,E2 21156.768} C_VEL
LIN {X 0,Y 424.118,Z 1218.33,A -85,B 0,C 180,E1 21154.189,E2 21154.189} C_VEL
LIN {X 0,Y 424.15,Z 1220.386,A -85,B 0,C 180,E1 21151.484,E2 21151.484} C_VEL
LIN {X 0,Y 424.132,Z 1220.933,A -85,B 0,C 180,E1 21148.918,E2 21148.918} C_VEL
LIN {X 0,Y 424.075,Z 1219.798,A -85,B 0,C 180,E1 21146.213,E2 21146.213} C_VEL
LIN {X 0,Y 424.032,Z 1216.958,A -85,B 0,C 180,E1 21143.363,E2 21143.363} C_VEL
LIN {X 0,Y 424.162,Z 1212.617,A -85,B 0,C 180,E1 21140.637,E2 21140.637} C_VEL
LIN {X 0,Y 424.586,Z 1206.557,A -85,B 0,C 180,E1 21137.9,E2 21137.9} C_VEL
LIN {X 0,Y 425.503,Z 1198.376,A -85,B 0,C 180,E1 21135.018,E2 21135.018} C_VEL
LIN {X 0,Y 426.943,Z 1188.686,A -85,B 0,C 180,E1 21132.273,E2 21132.273} C_VEL
LIN {X 0,Y 428.881,Z 1177.522,A -85,B 0,C 180,E1 21129.671,E2 21129.671} C_VEL
LIN {X 0,Y 431.488,Z 1164.412,A -85,B 0,C 180,E1 21127.087,E2 21127.087} C_VEL
LIN {X 0,Y 434.615,Z 1149.925,A -85,B 0,C 180,E1 21124.663,E2 21124.663} C_VEL
LIN {X 0,Y 438.44,Z 1133.027,A -85,B 0,C 180,E1 21122.273,E2 21122.273} C_VEL
LIN {X 0,Y 442.603,Z 1115.072,A -85,B 0,C 180,E1 21120.122,E2 21120.122} C_VEL
LIN {X 0,Y 447.356,Z 1094.813,A -85,B 0,C 180,E1 21118.06,E2 21118.06} C_VEL
LIN {X 0,Y 452.555,Z 1072.612,A -85,B 0,C 180,E1 21116.165,E2 21116.165} C_VEL
LIN {X 0,Y 457.724,Z 1050.167,A -85,B 0,C 180,E1 21114.572,E2 21114.572} C_VEL
LIN {X 0,Y 463.251,Z 1025.359,A -85,B 0,C 180,E1 21113.126,E2 21113.126} C_VEL
LIN {X 0,Y 468.462,Z 1000.947,A -85,B 0,C 180,E1 21111.99,E2 21111.99} C_VEL
LIN {X 0,Y 473.573,Z 974.805,A -85,B 0,C 180,E1 21111.037,E2 21111.037} C_VEL
LIN {X 0,Y 489.407,Z 881.612,A -85,B 0,C 180,E1 21108.379,E2 21108.379} C_VEL
LIN {X 0,Y 504.161,Z 810.755,A -85,B 0,C 180,E1 21106.394,E2 21106.394} C_VEL
LIN {X 0,Y 515.925,Z 761.241,A -85,B 0,C 180,E1 21105.047,E2 21105.047} C_VEL
LIN {X 0,Y 516.204,Z 759.816,A -85,B 0,C 180,E1 21104.215,E2 21104.215} C_VEL
LIN {X 0,Y 498.513,Z 834.403,A -85,B 0,C 180,E1 21102.179,E2 21102.179} C_VEL
LIN {X 0,Y 485.029,Z 901.645,A -85,B 0,C 180,E1 21100.283,E2 21100.283} C_VEL
LIN {X 0,Y 476.001,Z 954.839,A -85,B 0,C 180,E1 21098.728,E2 21098.728} C_VEL
LIN {X 0,Y 471.651,Z 978.572,A -85,B 0,C 180,E1 21097.785,E2 21097.785} C_VEL
LIN {X 0,Y 466.917,Z 1001.83,A -85,B 0,C 180,E1 21096.615,E2 21096.615} C_VEL
LIN {X 0,Y 461.999,Z 1024.241,A -85,B 0,C 180,E1 21095.227,E2 21095.227} C_VEL
LIN {X 0,Y 456.974,Z 1045.723,A -85,B 0,C 180,E1 21093.615,E2 21093.615} C_VEL
LIN {X 0,Y 451.955,Z 1066.16,A -85,B 0,C 180,E1 21091.775,E2 21091.775} C_VEL
LIN {X 0,Y 447.023,Z 1085.431,A -85,B 0,C 180,E1 21089.702,E2 21089.702} C_VEL
LIN {X 0,Y 442.418,Z 1102.909,A -85,B 0,C 180,E1 21087.457,E2 21087.457} C_VEL
LIN {X 0,Y 438.532,Z 1117.454,A -85,B 0,C 180,E1 21085.24,E2 21085.24} C_VEL
LIN {X 0,Y 434.929,Z 1131.06,A -85,B 0,C 180,E1 21082.794,E2 21082.794} C_VEL
LIN {X 0,Y 431.812,Z 1143.201,A -85,B 0,C 180,E1 21080.186,E2 21080.186} C_VEL
LIN {X 0,Y 429.409,Z 1153.149,A -85,B 0,C 180,E1 21077.623,E2 21077.623} C_VEL
LIN {X 0,Y 427.459,Z 1161.652,A -85,B 0,C 180,E1 21074.913,E2 21074.913} C_VEL
LIN {X 0,Y 426.005,Z 1168.76,A -85,B 0,C 180,E1 21072.06,E2 21072.06} C_VEL
LIN {X 0,Y 425.112,Z 1173.922,A -85,B 0,C 180,E1 21069.343,E2 21069.343} C_VEL
LIN {X 0,Y 424.556,Z 1177.59,A -85,B 0,C 180,E1 21066.494,E2 21066.494} C_VEL
LIN {X 0,Y 424.279,Z 1179.628,A -85,B 0,C 180,E1 21063.651,E2 21063.651} C_VEL
LIN {X 0,Y 424.171,Z 1180.127,A -85,B 0,C 180,E1 21060.948,E2 21060.948} C_VEL
LIN {X 0,Y 424.124,Z 1179.013,A -85,B 0,C 180,E1 21058.247,E2 21058.247} C_VEL
LIN {X 0,Y 424.168,Z 1176.282,A -85,B 0,C 180,E1 21055.406,E2 21055.406} C_VEL
LIN {X 0,Y 424.351,Z 1172.14,A -85,B 0,C 180,E1 21052.693,E2 21052.693} C_VEL
LIN {X 0,Y 424.739,Z 1166.243,A -85,B 0,C 180,E1 21049.971,E2 21049.971} C_VEL
LIN {X 0,Y 425.479,Z 1158.216,A -85,B 0,C 180,E1 21047.103,E2 21047.103} C_VEL
LIN {X 0,Y 426.556,Z 1149.004,A -85,B 0,C 180,E1 21044.459,E2 21044.459} C_VEL
LIN {X 0,Y 428.03,Z 1138.169,A -85,B 0,C 180,E1 21041.903,E2 21041.903} C_VEL
LIN {X 0,Y 429.9,Z 1125.687,A -85,B 0,C 180,E1 21039.442,E2 21039.442} C_VEL
LIN {X 0,Y 432.247,Z 1110.956,A -85,B 0,C 180,E1 21036.991,E2 21036.991} C_VEL
LIN {X 0,Y 434.78,Z 1095.622,A -85,B 0,C 180,E1 21034.824,E2 21034.824} C_VEL
LIN {X 0,Y 437.666,Z 1078.022,A -85,B 0,C 180,E1 21032.713,E2 21032.713} C_VEL
LIN {X 0,Y 440.555,Z 1059.749,A -85,B 0,C 180,E1 21030.871,E2 21030.871} C_VEL
LIN {X 0,Y 443.467,Z 1040.274,A -85,B 0,C 180,E1 21029.211,E2 21029.211} C_VEL
LIN {X 0,Y 446.429,Z 1018.885,A -85,B 0,C 180,E1 21027.69,E2 21027.69} C_VEL
LIN {X 0,Y 448.984,Z 998.255,A -85,B 0,C 180,E1 21026.479,E2 21026.479} C_VEL
LIN {X 0,Y 451.404,Z 975.872,A -85,B 0,C 180,E1 21025.42,E2 21025.42} C_VEL
LIN {X 0,Y 453.404,Z 952.932,A -85,B 0,C 180,E1 21024.588,E2 21024.588} C_VEL
LIN {X 0,Y 454.928,Z 930.048,A -85,B 0,C 180,E1 21023.982,E2 21023.982} C_VEL
LIN {X 0,Y 466.387,Z 717.953,A -85,B 0,C 180,E1 21019.727,E2 21019.727} C_VEL
LIN {X 0,Y 447.633,Z 684.334,A -85,B 0,C 180,E1 21017.253,E2 21017.253} C_VEL
LIN {X 0,Y 430.751,Z 655.876,A -85,B 0,C 180,E1 21014.861,E2 21014.861} C_VEL
LIN {X 0,Y 428.079,Z 651.453,A -85,B 0,C 180,E1 21014.464,E2 21014.464} C_VEL
LIN {X 0,Y 426.56,Z 648.067,A -85,B 0,C 180,E1 21014.208,E2 21014.208} C_VEL
LIN {X 0,Y 426.477,Z 647.541,A -85,B 0,C 180,E1 21014.163,E2 21014.163} C_VEL
LIN {X 0,Y 426.442,Z 647.546,A -85,B 0,C 180,E1 21010.362,E2 21010.362} C_VEL
LIN {X 0,Y 426.444,Z 647.55,A -85,B 0,C 180,E1 21006.554,E2 21006.554} C_VEL
LIN {X 0,Y 426.469,Z 647.541,A -85,B 0,C 180,E1 21002.794,E2 21002.794} C_VEL
LIN {X 0,Y 426.485,Z 647.54,A -85,B 0,C 180,E1 20999.023,E2 20999.023} C_VEL
LIN {X 0,Y 426.462,Z 647.545,A -85,B 0,C 180,E1 20995.183,E2 20995.183} C_VEL
LIN {X 0,Y 426.447,Z 647.545,A -85,B 0,C 180,E1 20991.444,E2 20991.444} C_VEL
LIN {X 0,Y 426.474,Z 647.537,A -85,B 0,C 180,E1 20987.606,E2 20987.606} C_VEL
LIN {X 0,Y 426.481,Z 647.531,A -85,B 0,C 180,E1 20983.837,E2 20983.837} C_VEL
LIN {X 0,Y 426.459,Z 647.542,A -85,B 0,C 180,E1 20979.993,E2 20979.993} C_VEL
LIN {X 0,Y 426.428,Z 647.55,A -85,B 0,C 180,E1 20976.194,E2 20976.194} C_VEL
LIN {X 0,Y 426.406,Z 647.536,A -85,B 0,C 180,E1 20972.286,E2 20972.286} C_VEL
LIN {X 0,Y 426.45,Z 647.544,A -85,B 0,C 180,E1 20968.524,E2 20968.524} C_VEL
LIN {X 0,Y 426.477,Z 647.532,A -85,B 0,C 180,E1 20964.756,E2 20964.756} C_VEL
LIN {X 0,Y 426.46,Z 647.541,A -85,B 0,C 180,E1 20961.1,E2 20961.1} C_VEL
LIN {X 0,Y 426.416,Z 647.538,A -85,B 0,C 180,E1 20957.406,E2 20957.406} C_VEL
LIN {X 0,Y 426.415,Z 647.548,A -85,B 0,C 180,E1 20953.519,E2 20953.519} C_VEL
LIN {X 0,Y 426.454,Z 647.544,A -85,B 0,C 180,E1 20949.684,E2 20949.684} C_VEL
LIN {X 0,Y 426.479,Z 647.541,A -85,B 0,C 180,E1 20945.927,E2 20945.927} C_VEL
LIN {X 0,Y 426.473,Z 647.542,A -85,B 0,C 180,E1 20944.546,E2 20944.546} C_VEL
LIN {X 0,Y 425.525,Z 647.664,A -85,B 0,C 180,E1 20943.512,E2 20943.512} C_VEL
LIN {X 0,Y 420.629,Z 648.274,A -85,B 0,C 180,E1 20941.414,E2 20941.414} C_VEL
LIN {X 0,Y 418.639,Z 648.523,A -85,B 0,C 180,E1 20940.142,E2 20940.142} C_VEL
LIN {X 0,Y 418.519,Z 648.536,A -85,B 0,C 180,E1 20939.836,E2 20939.836} C_VEL
LIN {X 0,Y 418.512,Z 648.537,A -85,B 0,C 180,E1 20935.993,E2 20935.993} C_VEL
LIN {X 0,Y 418.547,Z 648.532,A -85,B 0,C 180,E1 20932.127,E2 20932.127} C_VEL
LIN {X 0,Y 418.548,Z 648.65,A -85,B 0,C 180,E1 20929.396,E2 20929.396} C_VEL
LIN {X 0,Y 426.683,Z 674.529,A -85,B 0,C 180,E1 20926.389,E2 20926.389} C_VEL
LIN {X 0,Y 433.548,Z 699.333,A -85,B 0,C 180,E1 20923.627,E2 20923.627} C_VEL
LIN {X 0,Y 431.419,Z 741.595,A -85,B 0,C 180,E1 20919.858,E2 20919.858} C_VEL
LIN {X 0,Y 429.241,Z 784.156,A -85,B 0,C 180,E1 20916.073,E2 20916.073} C_VEL
LIN {X 0,Y 427.033,Z 829.401,A -85,B 0,C 180,E1 20912.052,E2 20912.052} C_VEL
LIN {X 0,Y 426.444,Z 844.53,A -85,B 0,C 180,E1 20910.748,E2 20910.748} C_VEL
LIN {X 0,Y 423.066,Z 984.859,A -85,B 0,C 180,E1 20907.735,E2 20907.735} C_VEL
LIN {X 0,Y 422.785,Z 1002.574,A -85,B 0,C 180,E1 20907.154,E2 20907.154} C_VEL
LIN {X 0,Y 422.267,Z 1018.937,A -85,B 0,C 180,E1 20906.354,E2 20906.354} C_VEL
LIN {X 0,Y 421.648,Z 1034.323,A -85,B 0,C 180,E1 20905.351,E2 20905.351} C_VEL
LIN {X 0,Y 420.86,Z 1049.812,A -85,B 0,C 180,E1 20904.041,E2 20904.041} C_VEL
LIN {X 0,Y 420.114,Z 1062.608,A -85,B 0,C 180,E1 20902.675,E2 20902.675} C_VEL
LIN {X 0,Y 419.351,Z 1075.115,A -85,B 0,C 180,E1 20901.026,E2 20901.026} C_VEL
LIN {X 0,Y 418.687,Z 1085.866,A -85,B 0,C 180,E1 20899.239,E2 20899.239} C_VEL
LIN {X 0,Y 418.209,Z 1094.786,A -85,B 0,C 180,E1 20897.386,E2 20897.386} C_VEL
LIN {X 0,Y 417.864,Z 1102.63,A -85,B 0,C 180,E1 20895.257,E2 20895.257} C_VEL
LIN {X 0,Y 417.719,Z 1107.975,A -85,B 0,C 180,E1 20893.282,E2 20893.282} C_VEL
LIN {X 0,Y 417.76,Z 1112.044,A -85,B 0,C 180,E1 20891.036,E2 20891.036} C_VEL
LIN {X 0,Y 417.989,Z 1114.003,A -85,B 0,C 180,E1 20888.92,E2 20888.92} C_VEL
LIN {X 0,Y 418.444,Z 1114.194,A -85,B 0,C 180,E1 20886.721,E2 20886.721} C_VEL
LIN {X 0,Y 419.096,Z 1112.613,A -85,B 0,C 180,E1 20884.65,E2 20884.65} C_VEL
LIN {X 0,Y 420.069,Z 1109.003,A -85,B 0,C 180,E1 20882.453,E2 20882.453} C_VEL
LIN {X 0,Y 421.174,Z 1104.109,A -85,B 0,C 180,E1 20880.541,E2 20880.541} C_VEL
LIN {X 0,Y 422.636,Z 1096.883,A -85,B 0,C 180,E1 20878.506,E2 20878.506} C_VEL
LIN {X 0,Y 424.151,Z 1088.73,A -85,B 0,C 180,E1 20876.754,E2 20876.754} C_VEL
LIN {X 0,Y 425.862,Z 1078.373,A -85,B 0,C 180,E1 20875.013,E2 20875.013} C_VEL
LIN {X 0,Y 427.531,Z 1066.881,A -85,B 0,C 180,E1 20873.484,E2 20873.484} C_VEL
LIN {X 0,Y 429.225,Z 1053.175,A -85,B 0,C 180,E1 20872.03,E2 20872.03} C_VEL
LIN {X 0,Y 430.646,Z 1038.913,A -85,B 0,C 180,E1 20870.846,E2 20870.846} C_VEL
LIN {X 0,Y 431.671,Z 1025.649,A -85,B 0,C 180,E1 20869.993,E2 20869.993} C_VEL
LIN {X 0,Y 432.438,Z 1012.765,A -85,B 0,C 180,E1 20869.338,E2 20869.338} C_VEL
LIN {X 0,Y 433.006,Z 998.161,A -85,B 0,C 180,E1 20868.775,E2 20868.775} C_VEL
LIN {X 0,Y 434.342,Z 958.419,A -85,B 0,C 180,E1 20867.766,E2 20867.766} C_VEL
LIN {X 0,Y 440.311,Z 857.996,A -85,B 0,C 180,E1 20865.317,E2 20865.317} C_VEL
LIN {X 0,Y 443.407,Z 822.236,A -85,B 0,C 180,E1 20862.095,E2 20862.095} C_VEL
LIN {X 0,Y 447.712,Z 775.855,A -85,B 0,C 180,E1 20857.892,E2 20857.892} C_VEL
LIN {X 0,Y 452.474,Z 730.353,A -85,B 0,C 180,E1 20853.768,E2 20853.768} C_VEL
LIN {X 0,Y 453.661,Z 718.887,A -85,B 0,C 180,E1 20852.711,E2 20852.711} C_VEL
LIN {X 0,Y 450.706,Z 707.186,A -85,B 0,C 180,E1 20850.784,E2 20850.784} C_VEL
LIN {X 0,Y 447.221,Z 697.107,A -85,B 0,C 180,E1 20848.752,E2 20848.752} C_VEL
LIN {X 0,Y 444.327,Z 690.031,A -85,B 0,C 180,E1 20847.001,E2 20847.001} C_VEL
LIN {X 0,Y 442.348,Z 685.822,A -85,B 0,C 180,E1 20845.745,E2 20845.745} C_VEL
LIN {X 0,Y 440.881,Z 682.479,A -85,B 0,C 180,E1 20844.665,E2 20844.665} C_VEL
LIN {X 0,Y 438.761,Z 678.134,A -85,B 0,C 180,E1 20842.898,E2 20842.898} C_VEL
LIN {X 0,Y 436.997,Z 674.973,A -85,B 0,C 180,E1 20841.069,E2 20841.069} C_VEL
LIN {X 0,Y 436.551,Z 673.412,A -85,B 0,C 180,E1 20840.278,E2 20840.278} C_VEL
LIN {X 0,Y 435.326,Z 672.465,A -85,B 0,C 180,E1 20838.481,E2 20838.481} C_VEL
LIN {X 0,Y 433.472,Z 675.955,A -85,B 0,C 180,E1 20837.116,E2 20837.116} C_VEL
LIN {X 0,Y 432.089,Z 679.656,A -85,B 0,C 180,E1 20835.834,E2 20835.834} C_VEL
LIN {X 0,Y 431.601,Z 681.901,A -85,B 0,C 180,E1 20835.389,E2 20835.389} C_VEL
LIN {X 0,Y 447.747,Z 713.357,A -85,B 0,C 180,E1 20832.997,E2 20832.997} C_VEL
LIN {X 0,Y 459.246,Z 737.398,A -85,B 0,C 180,E1 20831.378,E2 20831.378} C_VEL
LIN {X 0,Y 460.106,Z 744.187,A -85,B 0,C 180,E1 20831.134,E2 20831.134} C_VEL
LIN {X 0,Y 446.624,Z 979.792,A -85,B 0,C 180,E1 20826.272,E2 20826.272} C_VEL
LIN {X 0,Y 444.481,Z 1003.752,A -85,B 0,C 180,E1 20825.544,E2 20825.544} C_VEL
LIN {X 0,Y 441.964,Z 1026.695,A -85,B 0,C 180,E1 20824.598,E2 20824.598} C_VEL
LIN {X 0,Y 439.256,Z 1048.027,A -85,B 0,C 180,E1 20823.482,E2 20823.482} C_VEL
LIN {X 0,Y 436.259,Z 1069.221,A -85,B 0,C 180,E1 20822.12,E2 20822.12} C_VEL
LIN {X 0,Y 433.239,Z 1089.082,A -85,B 0,C 180,E1 20820.583,E2 20820.583} C_VEL
LIN {X 0,Y 430.076,Z 1108.709,A -85,B 0,C 180,E1 20818.765,E2 20818.765} C_VEL
LIN {X 0,Y 427.128,Z 1126.505,A -85,B 0,C 180,E1 20816.801,E2 20816.801} C_VEL
LIN {X 0,Y 424.37,Z 1143.126,A -85,B 0,C 180,E1 20814.646,E2 20814.646} C_VEL
LIN {X 0,Y 422.045,Z 1157.785,A -85,B 0,C 180,E1 20812.42,E2 20812.42} C_VEL
LIN {X 0,Y 420.062,Z 1171.113,A -85,B 0,C 180,E1 20810.043,E2 20810.043} C_VEL
LIN {X 0,Y 418.475,Z 1183,A -85,B 0,C 180,E1 20807.519,E2 20807.519} C_VEL
LIN {X 0,Y 417.258,Z 1194.007,A -85,B 0,C 180,E1 20804.713,E2 20804.713} C_VEL
LIN {X 0,Y 416.559,Z 1202.549,A -85,B 0,C 180,E1 20802.052,E2 20802.052} C_VEL
LIN {X 0,Y 416.214,Z 1209.247,A -85,B 0,C 180,E1 20799.4,E2 20799.4} C_VEL
LIN {X 0,Y 416.108,Z 1214.556,A -85,B 0,C 180,E1 20796.621,E2 20796.621} C_VEL
LIN {X 0,Y 416.135,Z 1218.064,A -85,B 0,C 180,E1 20793.994,E2 20793.994} C_VEL
LIN {X 0,Y 416.164,Z 1219.953,A -85,B 0,C 180,E1 20791.375,E2 20791.375} C_VEL
LIN {X 0,Y 416.138,Z 1220.489,A -85,B 0,C 180,E1 20788.759,E2 20788.759} C_VEL
LIN {X 0,Y 416.076,Z 1219.337,A -85,B 0,C 180,E1 20786.002,E2 20786.002} C_VEL
LIN {X 0,Y 416.035,Z 1216.484,A -85,B 0,C 180,E1 20783.096,E2 20783.096} C_VEL
LIN {X 0,Y 416.191,Z 1212.124,A -85,B 0,C 180,E1 20780.317,E2 20780.317} C_VEL
LIN {X 0,Y 416.68,Z 1206.056,A -85,B 0,C 180,E1 20777.526,E2 20777.526} C_VEL
LIN {X 0,Y 417.695,Z 1197.872,A -85,B 0,C 180,E1 20774.589,E2 20774.589} C_VEL
LIN {X 0,Y 419.272,Z 1188.186,A -85,B 0,C 180,E1 20771.794,E2 20771.794} C_VEL
LIN {X 0,Y 421.379,Z 1177.056,A -85,B 0,C 180,E1 20769.148,E2 20769.148} C_VEL
LIN {X 0,Y 424.356,Z 1163.258,A -85,B 0,C 180,E1 20766.385,E2 20766.385} C_VEL
LIN {X 0,Y 427.749,Z 1148.725,A -85,B 0,C 180,E1 20763.929,E2 20763.929} C_VEL
LIN {X 0,Y 431.865,Z 1131.884,A -85,B 0,C 180,E1 20761.512,E2 20761.512} C_VEL
LIN {X 0,Y 436.492,Z 1113.442,A -85,B 0,C 180,E1 20759.279,E2 20759.279} C_VEL
LIN {X 0,Y 441.521,Z 1093.491,A -85,B 0,C 180,E1 20757.23,E2 20757.23} C_VEL
LIN {X 0,Y 446.951,Z 1072.009,A -85,B 0,C 180,E1 20755.372,E2 20755.372} C_VEL
LIN {X 0,Y 452.716,Z 1048.9,A -85,B 0,C 180,E1 20753.705,E2 20753.705} C_VEL
LIN {X 0,Y 458.533,Z 1024.948,A -85,B 0,C 180,E1 20752.289,E2 20752.289} C_VEL
LIN {X 0,Y 464.036,Z 1001.392,A -85,B 0,C 180,E1 20751.167,E2 20751.167} C_VEL
LIN {X 0,Y 469.665,Z 975.165,A -85,B 0,C 180,E1 20750.186,E2 20750.186} C_VEL
LIN {X 0,Y 487.33,Z 880.913,A -85,B 0,C 180,E1 20747.442,E2 20747.442} C_VEL
LIN {X 0,Y 503.715,Z 808.69,A -85,B 0,C 180,E1 20745.415,E2 20745.415} C_VEL
LIN {X 0,Y 511.12,Z 779.254,A -85,B 0,C 180,E1 20744.614,E2 20744.614} C_VEL
LIN {X 0,Y 493.42,Z 851.072,A -85,B 0,C 180,E1 20742.638,E2 20742.638} C_VEL
LIN {X 0,Y 479.732,Z 916.139,A -85,B 0,C 180,E1 20740.782,E2 20740.782} C_VEL
LIN {X 0,Y 472.251,Z 956.671,A -85,B 0,C 180,E1 20739.554,E2 20739.554} C_VEL
LIN {X 0,Y 467.412,Z 980.486,A -85,B 0,C 180,E1 20738.58,E2 20738.58} C_VEL
LIN {X 0,Y 462.389,Z 1002.942,A -85,B 0,C 180,E1 20737.422,E2 20737.422} C_VEL
LIN {X 0,Y 456.936,Z 1025.589,A -85,B 0,C 180,E1 20735.985,E2 20735.985} C_VEL
LIN {X 0,Y 451.403,Z 1047.274,A -85,B 0,C 180,E1 20734.317,E2 20734.317} C_VEL
LIN {X 0,Y 446.086,Z 1067.278,A -85,B 0,C 180,E1 20732.471,E2 20732.471} C_VEL
LIN {X 0,Y 440.847,Z 1086.269,A -85,B 0,C 180,E1 20730.386,E2 20730.386} C_VEL
LIN {X 0,Y 436.084,Z 1103.089,A -85,B 0,C 180,E1 20728.188,E2 20728.188} C_VEL
LIN {X 0,Y 431.914,Z 1117.58,A -85,B 0,C 180,E1 20725.95,E2 20725.95} C_VEL
LIN {X 0,Y 427.949,Z 1131.519,A -85,B 0,C 180,E1 20723.406,E2 20723.406} C_VEL
LIN {X 0,Y 424.643,Z 1143.454,A -85,B 0,C 180,E1 20720.802,E2 20720.802} C_VEL
LIN {X 0,Y 421.931,Z 1153.78,A -85,B 0,C 180,E1 20718.089,E2 20718.089} C_VEL
LIN {X 0,Y 419.728,Z 1162.625,A -85,B 0,C 180,E1 20715.194,E2 20715.194} C_VEL
LIN {X 0,Y 418.173,Z 1169.59,A -85,B 0,C 180,E1 20712.29,E2 20712.29} C_VEL
LIN {X 0,Y 417.167,Z 1174.82,A -85,B 0,C 180,E1 20709.383,E2 20709.383} C_VEL
LIN {X 0,Y 416.587,Z 1178.37,A -85,B 0,C 180,E1 20706.48,E2 20706.48} C_VEL
LIN {X 0,Y 416.3,Z 1180.146,A -85,B 0,C 180,E1 20703.721,E2 20703.721} C_VEL
LIN {X 0,Y 416.175,Z 1180.493,A -85,B 0,C 180,E1 20700.829,E2 20700.829} C_VEL
LIN {X 0,Y 416.132,Z 1179.352,A -85,B 0,C 180,E1 20698.213,E2 20698.213} C_VEL
LIN {X 0,Y 416.178,Z 1176.498,A -85,B 0,C 180,E1 20695.318,E2 20695.318} C_VEL
LIN {X 0,Y 416.371,Z 1172.244,A -85,B 0,C 180,E1 20692.552,E2 20692.552} C_VEL
LIN {X 0,Y 416.786,Z 1166.244,A -85,B 0,C 180,E1 20689.777,E2 20689.777} C_VEL
LIN {X 0,Y 417.519,Z 1158.496,A -85,B 0,C 180,E1 20686.994,E2 20686.994} C_VEL
LIN {X 0,Y 418.649,Z 1149.089,A -85,B 0,C 180,E1 20684.266,E2 20684.266} C_VEL
LIN {X 0,Y 420.254,Z 1137.718,A -85,B 0,C 180,E1 20681.556,E2 20681.556} C_VEL
LIN {X 0,Y 422.214,Z 1125.032,A -85,B 0,C 180,E1 20679.051,E2 20679.051} C_VEL
LIN {X 0,Y 424.517,Z 1110.962,A -85,B 0,C 180,E1 20676.694,E2 20676.694} C_VEL
LIN {X 0,Y 427.216,Z 1094.997,A -85,B 0,C 180,E1 20674.421,E2 20674.421} C_VEL
LIN {X 0,Y 430.113,Z 1077.81,A -85,B 0,C 180,E1 20672.342,E2 20672.342} C_VEL
LIN {X 0,Y 433.204,Z 1058.777,A -85,B 0,C 180,E1 20670.404,E2 20670.404} C_VEL
LIN {X 0,Y 436.197,Z 1039.203,A -85,B 0,C 180,E1 20668.733,E2 20668.733} C_VEL
LIN {X 0,Y 439.144,Z 1018.319,A -85,B 0,C 180,E1 20667.242,E2 20667.242} C_VEL
LIN {X 0,Y 441.917,Z 996.222,A -85,B 0,C 180,E1 20665.949,E2 20665.949} C_VEL
LIN {X 0,Y 444.337,Z 974.031,A -85,B 0,C 180,E1 20664.908,E2 20664.908} C_VEL
LIN {X 0,Y 446.393,Z 950.913,A -85,B 0,C 180,E1 20664.07,E2 20664.07} C_VEL
LIN {X 0,Y 447.972,Z 927.031,A -85,B 0,C 180,E1 20663.455,E2 20663.455} C_VEL
LIN {X 0,Y 459.572,Z 720.749,A -85,B 0,C 180,E1 20659.245,E2 20659.245} C_VEL
LIN {X 0,Y 441.132,Z 687.752,A -85,B 0,C 180,E1 20656.758,E2 20656.758} C_VEL
LIN {X 0,Y 425.176,Z 660.777,A -85,B 0,C 180,E1 20654.446,E2 20654.446} C_VEL
LIN {X 0,Y 420.391,Z 652.748,A -85,B 0,C 180,E1 20653.707,E2 20653.707} C_VEL
LIN {X 0,Y 418.675,Z 649.434,A -85,B 0,C 180,E1 20653.424,E2 20653.424} C_VEL
LIN {X 0,Y 418.508,Z 648.54,A -85,B 0,C 180,E1 20653.343,E2 20653.343} C_VEL
LIN {X 0,Y 418.484,Z 648.538,A -85,B 0,C 180,E1 20649.641,E2 20649.641} C_VEL
LIN {X 0,Y 418.52,Z 648.532,A -85,B 0,C 180,E1 20645.828,E2 20645.828} C_VEL
LIN {X 0,Y 418.546,Z 648.528,A -85,B 0,C 180,E1 20642.004,E2 20642.004} C_VEL
LIN {X 0,Y 418.531,Z 648.537,A -85,B 0,C 180,E1 20638.178,E2 20638.178} C_VEL
LIN {X 0,Y 418.493,Z 648.542,A -85,B 0,C 180,E1 20634.417,E2 20634.417} C_VEL
LIN {X 0,Y 418.469,Z 648.543,A -85,B 0,C 180,E1 20630.516,E2 20630.516} C_VEL
LIN {X 0,Y 418.506,Z 648.534,A -85,B 0,C 180,E1 20626.662,E2 20626.662} C_VEL
LIN {X 0,Y 418.533,Z 648.522,A -85,B 0,C 180,E1 20622.839,E2 20622.839} C_VEL
LIN {X 0,Y 418.544,Z 648.521,A -85,B 0,C 180,E1 20618.935,E2 20618.935} C_VEL
LIN {X 0,Y 418.516,Z 648.539,A -85,B 0,C 180,E1 20615.211,E2 20615.211} C_VEL
LIN {X 0,Y 418.526,Z 648.527,A -85,B 0,C 180,E1 20611.097,E2 20611.097} C_VEL
LIN {X 0,Y 418.541,Z 648.519,A -85,B 0,C 180,E1 20607.263,E2 20607.263} C_VEL
LIN {X 0,Y 418.53,Z 648.533,A -85,B 0,C 180,E1 20603.417,E2 20603.417} C_VEL
LIN {X 0,Y 418.498,Z 648.518,A -85,B 0,C 180,E1 20599.54,E2 20599.54} C_VEL
LIN {X 0,Y 418.463,Z 648.539,A -85,B 0,C 180,E1 20595.613,E2 20595.613} C_VEL
LIN {X 0,Y 418.498,Z 648.536,A -85,B 0,C 180,E1 20591.619,E2 20591.619} C_VEL
LIN {X 0,Y 418.529,Z 648.534,A -85,B 0,C 180,E1 20587.825,E2 20587.825} C_VEL
LIN {X 0,Y 418.546,Z 648.53,A -85,B 0,C 180,E1 20583.919,E2 20583.919} C_VEL
LIN {X 0,Y 418.543,Z 648.534,A -85,B 0,C 180,E1 20580.049,E2 20580.049} C_VEL
LIN {X 0,Y 418.519,Z 648.536,A -85,B 0,C 180,E1 20579.836,E2 20579.836} C_VEL
LIN {X 0,Y 417.459,Z 648.668,A -85,B 0,C 180,E1 20578.782,E2 20578.782} C_VEL
LIN {X 0,Y 410.962,Z 649.479,A -85,B 0,C 180,E1 20575.734,E2 20575.734} C_VEL
LIN {X 0,Y 410.545,Z 649.53,A -85,B 0,C 180,E1 20575.035,E2 20575.035} C_VEL
LIN {X 0,Y 410.579,Z 649.526,A -85,B 0,C 180,E1 20571.19,E2 20571.19} C_VEL
LIN {X 0,Y 410.629,Z 649.683,A -85,B 0,C 180,E1 20569.865,E2 20569.865} C_VEL
LIN {X 0,Y 419.307,Z 677.177,A -85,B 0,C 180,E1 20566.628,E2 20566.628} C_VEL
LIN {X 0,Y 426.045,Z 701.555,A -85,B 0,C 180,E1 20563.884,E2 20563.884} C_VEL
LIN {X 0,Y 423.748,Z 744.509,A -85,B 0,C 180,E1 20560.005,E2 20560.005} C_VEL
LIN {X 0,Y 421.469,Z 787.96,A -85,B 0,C 180,E1 20556.108,E2 20556.108} C_VEL
LIN {X 0,Y 419.196,Z 833.086,A -85,B 0,C 180,E1 20552.071,E2 20552.071} C_VEL
LIN {X 0,Y 418.699,Z 845.277,A -85,B 0,C 180,E1 20551.015,E2 20551.015} C_VEL
LIN {X 0,Y 415.197,Z 984.988,A -85,B 0,C 180,E1 20547.931,E2 20547.931} C_VEL
LIN {X 0,Y 414.899,Z 1003.263,A -85,B 0,C 180,E1 20547.325,E2 20547.325} C_VEL
LIN {X 0,Y 414.366,Z 1019.687,A -85,B 0,C 180,E1 20546.51,E2 20546.51} C_VEL
LIN {X 0,Y 413.725,Z 1035.271,A -85,B 0,C 180,E1 20545.476,E2 20545.476} C_VEL
LIN {X 0,Y 412.924,Z 1050.654,A -85,B 0,C 180,E1 20544.153,E2 20544.153} C_VEL
LIN {X 0,Y 412.125,Z 1064.089,A -85,B 0,C 180,E1 20542.687,E2 20542.687} C_VEL
LIN {X 0,Y 411.367,Z 1076.279,A -85,B 0,C 180,E1 20541.042,E2 20541.042} C_VEL
LIN {X 0,Y 410.684,Z 1087.351,A -85,B 0,C 180,E1 20539.159,E2 20539.159} C_VEL
LIN {X 0,Y 410.214,Z 1096.05,A -85,B 0,C 180,E1 20537.296,E2 20537.296} C_VEL
LIN {X 0,Y 409.88,Z 1103.868,A -85,B 0,C 180,E1 20535.127,E2 20535.127} C_VEL
LIN {X 0,Y 409.749,Z 1109.119,A -85,B 0,C 180,E1 20533.114,E2 20533.114} C_VEL
LIN {X 0,Y 409.806,Z 1112.955,A -85,B 0,C 180,E1 20530.968,E2 20530.968} C_VEL
LIN {X 0,Y 410.059,Z 1114.995,A -85,B 0,C 180,E1 20528.833,E2 20528.833} C_VEL
LIN {X 0,Y 410.555,Z 1115.258,A -85,B 0,C 180,E1 20526.57,E2 20526.57} C_VEL
LIN {X 0,Y 411.261,Z 1113.749,A -85,B 0,C 180,E1 20524.459,E2 20524.459} C_VEL
LIN {X 0,Y 412.304,Z 1110.194,A -85,B 0,C 180,E1 20522.221,E2 20522.221} C_VEL
LIN {X 0,Y 413.494,Z 1105.406,A -85,B 0,C 180,E1 20520.274,E2 20520.274} C_VEL
LIN {X 0,Y 415.053,Z 1098.247,A -85,B 0,C 180,E1 20518.202,E2 20518.202} C_VEL
LIN {X 0,Y 416.662,Z 1090.161,A -85,B 0,C 180,E1 20516.42,E2 20516.42} C_VEL
LIN {X 0,Y 418.469,Z 1079.863,A -85,B 0,C 180,E1 20514.65,E2 20514.65} C_VEL
LIN {X 0,Y 420.257,Z 1068.572,A -85,B 0,C 180,E1 20513.096,E2 20513.096} C_VEL
LIN {X 0,Y 422.053,Z 1055.026,A -85,B 0,C 180,E1 20511.619,E2 20511.619} C_VEL
LIN {X 0,Y 423.554,Z 1040.944,A -85,B 0,C 180,E1 20510.417,E2 20510.417} C_VEL
LIN {X 0,Y 424.639,Z 1027.928,A -85,B 0,C 180,E1 20509.551,E2 20509.551} C_VEL
LIN {X 0,Y 425.512,Z 1014.776,A -85,B 0,C 180,E1 20508.853,E2 20508.853} C_VEL
LIN {X 0,Y 426.178,Z 1000.064,A -85,B 0,C 180,E1 20508.258,E2 20508.258} C_VEL
LIN {X 0,Y 427.551,Z 961.579,A -85,B 0,C 180,E1 20507.242,E2 20507.242} C_VEL
LIN {X 0,Y 433.931,Z 859.431,A -85,B 0,C 180,E1 20504.699,E2 20504.699} C_VEL
LIN {X 0,Y 437.689,Z 819.711,A -85,B 0,C 180,E1 20501.068,E2 20501.068} C_VEL
LIN {X 0,Y 441.927,Z 777.142,A -85,B 0,C 180,E1 20497.165,E2 20497.165} C_VEL
LIN {X 0,Y 447.155,Z 731.925,A -85,B 0,C 180,E1 20493.001,E2 20493.001} C_VEL
LIN {X 0,Y 448.251,Z 723.348,A -85,B 0,C 180,E1 20492.209,E2 20492.209} C_VEL
LIN {X 0,Y 445.459,Z 711.865,A -85,B 0,C 180,E1 20490.258,E2 20490.258} C_VEL
LIN {X 0,Y 442.467,Z 702.673,A -85,B 0,C 180,E1 20488.302,E2 20488.302} C_VEL
LIN {X 0,Y 439.934,Z 696.148,A -85,B 0,C 180,E1 20486.629,E2 20486.629} C_VEL
LIN {X 0,Y 437.211,Z 689.56,A -85,B 0,C 180,E1 20484.565,E2 20484.565} C_VEL
LIN {X 0,Y 435.352,Z 685.359,A -85,B 0,C 180,E1 20482.837,E2 20482.837} C_VEL
LIN {X 0,Y 433.582,Z 682.094,A -85,B 0,C 180,E1 20480.894,E2 20480.894} C_VEL
LIN {X 0,Y 433.247,Z 680.665,A -85,B 0,C 180,E1 20480.086,E2 20480.086} C_VEL
LIN {X 0,Y 432.409,Z 679.901,A -85,B 0,C 180,E1 20478.718,E2 20478.718} C_VEL
LIN {X 0,Y 430.679,Z 682.913,A -85,B 0,C 180,E1 20477.496,E2 20477.496} C_VEL
LIN {X 0,Y 429.282,Z 686.406,A -85,B 0,C 180,E1 20476.317,E2 20476.317} C_VEL
LIN {X 0,Y 428.037,Z 690.673,A -85,B 0,C 180,E1 20475.483,E2 20475.483} C_VEL
LIN {X 0,Y 443.992,Z 722.053,A -85,B 0,C 180,E1 20473.092,E2 20473.092} C_VEL
LIN {X 0,Y 452.832,Z 740.793,A -85,B 0,C 180,E1 20471.827,E2 20471.827} C_VEL
LIN {X 0,Y 453.329,Z 745.819,A -85,B 0,C 180,E1 20471.655,E2 20471.655} C_VEL
LIN {X 0,Y 439.435,Z 979.503,A -85,B 0,C 180,E1 20466.728,E2 20466.728} C_VEL
LIN {X 0,Y 437.213,Z 1003.636,A -85,B 0,C 180,E1 20465.98,E2 20465.98} C_VEL
LIN {X 0,Y 434.699,Z 1025.871,A -85,B 0,C 180,E1 20465.048,E2 20465.048} C_VEL
LIN {X 0,Y 431.912,Z 1047.379,A -85,B 0,C 180,E1 20463.909,E2 20463.909} C_VEL
LIN {X 0,Y 428.794,Z 1068.852,A -85,B 0,C 180,E1 20462.51,E2 20462.51} C_VEL
LIN {X 0,Y 425.701,Z 1088.668,A -85,B 0,C 180,E1 20460.954,E2 20460.954} C_VEL
LIN {X 0,Y 422.449,Z 1108.356,A -85,B 0,C 180,E1 20459.101,E2 20459.101} C_VEL
LIN {X 0,Y 419.39,Z 1126.322,A -85,B 0,C 180,E1 20457.086,E2 20457.086} C_VEL
LIN {X 0,Y 416.584,Z 1142.809,A -85,B 0,C 180,E1 20454.91,E2 20454.91} C_VEL
LIN {X 0,Y 414.124,Z 1157.894,A -85,B 0,C 180,E1 20452.573,E2 20452.573} C_VEL
LIN {X 0,Y 412.061,Z 1171.475,A -85,B 0,C 180,E1 20450.097,E2 20450.097} C_VEL
LIN {X 0,Y 410.411,Z 1183.637,A -85,B 0,C 180,E1 20447.435,E2 20447.435} C_VEL
LIN {X 0,Y 409.253,Z 1193.965,A -85,B 0,C 180,E1 20444.718,E2 20444.718} C_VEL
LIN {X 0,Y 408.552,Z 1202.434,A -85,B 0,C 180,E1 20442.005,E2 20442.005} C_VEL
LIN {X 0,Y 408.216,Z 1209.095,A -85,B 0,C 180,E1 20439.301,E2 20439.301} C_VEL
LIN {X 0,Y 408.121,Z 1214.32,A -85,B 0,C 180,E1 20436.469,E2 20436.469} C_VEL
LIN {X 0,Y 408.153,Z 1217.771,A -85,B 0,C 180,E1 20433.791,E2 20433.791} C_VEL
LIN {X 0,Y 408.182,Z 1219.574,A -85,B 0,C 180,E1 20431.121,E2 20431.121} C_VEL
LIN {X 0,Y 408.143,Z 1220.02,A -85,B 0,C 180,E1 20428.454,E2 20428.454} C_VEL
LIN {X 0,Y 408.074,Z 1218.879,A -85,B 0,C 180,E1 20425.781,E2 20425.781} C_VEL
LIN {X 0,Y 408.05,Z 1216.023,A -85,B 0,C 180,E1 20422.819,E2 20422.819} C_VEL
LIN {X 0,Y 408.228,Z 1211.649,A -85,B 0,C 180,E1 20419.983,E2 20419.983} C_VEL
LIN {X 0,Y 408.784,Z 1205.582,A -85,B 0,C 180,E1 20417.137,E2 20417.137} C_VEL
LIN {X 0,Y 409.845,Z 1197.864,A -85,B 0,C 180,E1 20414.286,E2 20414.286} C_VEL
LIN {X 0,Y 411.598,Z 1187.911,A -85,B 0,C 180,E1 20411.343,E2 20411.343} C_VEL
LIN {X 0,Y 413.923,Z 1176.671,A -85,B 0,C 180,E1 20408.605,E2 20408.605} C_VEL
LIN {X 0,Y 417.125,Z 1162.963,A -85,B 0,C 180,E1 20405.8,E2 20405.8} C_VEL
LIN {X 0,Y 420.769,Z 1148.572,A -85,B 0,C 180,E1 20403.311,E2 20403.311} C_VEL
LIN {X 0,Y 425.414,Z 1130.909,A -85,B 0,C 180,E1 20400.731,E2 20400.731} C_VEL
LIN {X 0,Y 430.52,Z 1112.043,A -85,B 0,C 180,E1 20398.416,E2 20398.416} C_VEL
LIN {X 0,Y 436.106,Z 1091.607,A -85,B 0,C 180,E1 20396.298,E2 20396.298} C_VEL
LIN {X 0,Y 442.128,Z 1069.583,A -85,B 0,C 180,E1 20394.383,E2 20394.383} C_VEL
LIN {X 0,Y 448.32,Z 1046.725,A -85,B 0,C 180,E1 20392.732,E2 20392.732} C_VEL
LIN {X 0,Y 454.541,Z 1023.192,A -85,B 0,C 180,E1 20391.336,E2 20391.336} C_VEL
LIN {X 0,Y 460.671,Z 999.026,A -85,B 0,C 180,E1 20390.184,E2 20390.184} C_VEL
LIN {X 0,Y 467.147,Z 971.135,A -85,B 0,C 180,E1 20389.152,E2 20389.152} C_VEL
LIN {X 0,Y 485.251,Z 882.877,A -85,B 0,C 180,E1 20386.56,E2 20386.56} C_VEL
LIN {X 0,Y 502.054,Z 813.845,A -85,B 0,C 180,E1 20384.613,E2 20384.613} C_VEL
LIN {X 0,Y 484.44,Z 884.891,A -85,B 0,C 180,E1 20382.622,E2 20382.622} C_VEL
LIN {X 0,Y 469.581,Z 955.653,A -85,B 0,C 180,E1 20380.52,E2 20380.52} C_VEL
LIN {X 0,Y 464.199,Z 979.826,A -85,B 0,C 180,E1 20379.535,E2 20379.535} C_VEL
LIN {X 0,Y 458.574,Z 1002.789,A -85,B 0,C 180,E1 20378.343,E2 20378.343} C_VEL
LIN {X 0,Y 452.634,Z 1025.367,A -85,B 0,C 180,E1 20376.899,E2 20376.899} C_VEL
LIN {X 0,Y 446.432,Z 1047.662,A -85,B 0,C 180,E1 20375.163,E2 20375.163} C_VEL
LIN {X 0,Y 440.537,Z 1068.106,A -85,B 0,C 180,E1 20373.242,E2 20373.242} C_VEL
LIN {X 0,Y 434.794,Z 1087.338,A -85,B 0,C 180,E1 20371.086,E2 20371.086} C_VEL
LIN {X 0,Y 429.6,Z 1104.395,A -85,B 0,C 180,E1 20368.805,E2 20368.805} C_VEL
LIN {X 0,Y 424.93,Z 1119.452,A -85,B 0,C 180,E1 20366.409,E2 20366.409} C_VEL
LIN {X 0,Y 420.743,Z 1133.091,A -85,B 0,C 180,E1 20363.831,E2 20363.831} C_VEL
LIN {X 0,Y 417.107,Z 1145.223,A -85,B 0,C 180,E1 20361.077,E2 20361.077} C_VEL
LIN {X 0,Y 414.227,Z 1155.361,A -85,B 0,C 180,E1 20358.291,E2 20358.291} C_VEL
LIN {X 0,Y 411.929,Z 1164.035,A -85,B 0,C 180,E1 20355.345,E2 20355.345} C_VEL
LIN {X 0,Y 410.287,Z 1170.744,A -85,B 0,C 180,E1 20352.387,E2 20352.387} C_VEL
LIN {X 0,Y 409.224,Z 1175.739,A -85,B 0,C 180,E1 20349.425,E2 20349.425} C_VEL
LIN {X 0,Y 408.614,Z 1179.114,A -85,B 0,C 180,E1 20346.466,E2 20346.466} C_VEL
LIN {X 0,Y 408.315,Z 1180.726,A -85,B 0,C 180,E1 20343.653,E2 20343.653} C_VEL
LIN {X 0,Y 408.178,Z 1180.857,A -85,B 0,C 180,E1 20340.705,E2 20340.705} C_VEL
LIN {X 0,Y 408.14,Z 1179.511,A -85,B 0,C 180,E1 20337.897,E2 20337.897} C_VEL
LIN {X 0,Y 408.196,Z 1176.522,A -85,B 0,C 180,E1 20335.085,E2 20335.085} C_VEL
LIN {X 0,Y 408.422,Z 1171.753,A -85,B 0,C 180,E1 20332.123,E2 20332.123} C_VEL
LIN {X 0,Y 408.894,Z 1165.549,A -85,B 0,C 180,E1 20329.293,E2 20329.293} C_VEL
LIN {X 0,Y 409.709,Z 1157.44,A -85,B 0,C 180,E1 20326.454,E2 20326.454} C_VEL
LIN {X 0,Y 410.905,Z 1147.934,A -85,B 0,C 180,E1 20323.753,E2 20323.753} C_VEL
LIN {X 0,Y 412.586,Z 1136.491,A -85,B 0,C 180,E1 20321.053,E2 20321.053} C_VEL
LIN {X 0,Y 414.675,Z 1123.589,A -85,B 0,C 180,E1 20318.503,E2 20318.503} C_VEL
LIN {X 0,Y 417.114,Z 1109.127,A -85,B 0,C 180,E1 20316.105,E2 20316.105} C_VEL
LIN {X 0,Y 419.853,Z 1093.239,A -85,B 0,C 180,E1 20313.863,E2 20313.863} C_VEL
LIN {X 0,Y 422.845,Z 1075.881,A -85,B 0,C 180,E1 20311.779,E2 20311.779} C_VEL
LIN {X 0,Y 425.876,Z 1057.676,A -85,B 0,C 180,E1 20309.92,E2 20309.92} C_VEL
LIN {X 0,Y 429.121,Z 1036.93,A -85,B 0,C 180,E1 20308.15,E2 20308.15} C_VEL
LIN {X 0,Y 431.97,Z 1016.943,A -85,B 0,C 180,E1 20306.734,E2 20306.734} C_VEL
LIN {X 0,Y 434.736,Z 995.284,A -85,B 0,C 180,E1 20305.467,E2 20305.467} C_VEL
LIN {X 0,Y 437.223,Z 972.784,A -85,B 0,C 180,E1 20304.412,E2 20304.412} C_VEL
LIN {X 0,Y 439.269,Z 950.067,A -85,B 0,C 180,E1 20303.586,E2 20303.586} C_VEL
LIN {X 0,Y 440.92,Z 925.924,A -85,B 0,C 180,E1 20302.961,E2 20302.961} C_VEL
LIN {X 0,Y 452.743,Z 723.497,A -85,B 0,C 180,E1 20298.741,E2 20298.741} C_VEL
LIN {X 0,Y 433.786,Z 689.659,A -85,B 0,C 180,E1 20296.13,E2 20296.13} C_VEL
LIN {X 0,Y 417.371,Z 661.875,A -85,B 0,C 180,E1 20293.676,E2 20293.676} C_VEL
LIN {X 0,Y 412.233,Z 653.513,A -85,B 0,C 180,E1 20292.874,E2 20292.874} C_VEL
LIN {X 0,Y 410.675,Z 650.18,A -85,B 0,C 180,E1 20292.6,E2 20292.6} C_VEL
LIN {X 0,Y 410.569,Z 649.522,A -85,B 0,C 180,E1 20292.544,E2 20292.544} C_VEL
LIN {X 0,Y 410.537,Z 649.533,A -85,B 0,C 180,E1 20288.753,E2 20288.753} C_VEL
LIN {X 0,Y 410.571,Z 649.52,A -85,B 0,C 180,E1 20284.85,E2 20284.85} C_VEL
LIN {X 0,Y 410.603,Z 649.525,A -85,B 0,C 180,E1 20280.92,E2 20280.92} C_VEL
LIN {X 0,Y 410.595,Z 649.524,A -85,B 0,C 180,E1 20277.091,E2 20277.091} C_VEL
LIN {X 0,Y 410.565,Z 649.525,A -85,B 0,C 180,E1 20273.239,E2 20273.239} C_VEL
LIN {X 0,Y 410.571,Z 649.523,A -85,B 0,C 180,E1 20269.344,E2 20269.344} C_VEL
LIN {X 0,Y 410.609,Z 649.519,A -85,B 0,C 180,E1 20265.539,E2 20265.539} C_VEL
LIN {X 0,Y 410.596,Z 649.522,A -85,B 0,C 180,E1 20261.663,E2 20261.663} C_VEL
LIN {X 0,Y 410.567,Z 649.515,A -85,B 0,C 180,E1 20257.84,E2 20257.84} C_VEL
LIN {X 0,Y 410.527,Z 649.526,A -85,B 0,C 180,E1 20254.052,E2 20254.052} C_VEL
LIN {X 0,Y 410.55,Z 649.526,A -85,B 0,C 180,E1 20250.141,E2 20250.141} C_VEL
LIN {X 0,Y 410.583,Z 649.504,A -85,B 0,C 180,E1 20246.232,E2 20246.232} C_VEL
LIN {X 0,Y 410.608,Z 649.522,A -85,B 0,C 180,E1 20242.305,E2 20242.305} C_VEL
LIN {X 0,Y 410.587,Z 649.499,A -85,B 0,C 180,E1 20238.483,E2 20238.483} C_VEL
LIN {X 0,Y 410.578,Z 649.527,A -85,B 0,C 180,E1 20234.609,E2 20234.609} C_VEL
LIN {X 0,Y 410.605,Z 649.52,A -85,B 0,C 180,E1 20230.662,E2 20230.662} C_VEL
LIN {X 0,Y 410.602,Z 649.518,A -85,B 0,C 180,E1 20226.768,E2 20226.768} C_VEL
LIN {X 0,Y 410.576,Z 649.524,A -85,B 0,C 180,E1 20222.911,E2 20222.911} C_VEL
LIN {X 0,Y 410.536,Z 649.53,A -85,B 0,C 180,E1 20219.009,E2 20219.009} C_VEL
LIN {X 0,Y 410.545,Z 649.53,A -85,B 0,C 180,E1 20215.035,E2 20215.035} C_VEL
LIN {X 0,Y 409.567,Z 649.653,A -85,B 0,C 180,E1 20214.32,E2 20214.32} C_VEL
LIN {X 0,Y 403.219,Z 650.443,A -85,B 0,C 180,E1 20212.372,E2 20212.372} C_VEL
LIN {X 0,Y 402.656,Z 650.511,A -85,B 0,C 180,E1 20211.843,E2 20211.843} C_VEL
LIN {X 0,Y 402.679,Z 650.57,A -85,B 0,C 180,E1 20210.384,E2 20210.384} C_VEL
LIN {X 0,Y 411.308,Z 677.726,A -85,B 0,C 180,E1 20207.107,E2 20207.107} C_VEL
LIN {X 0,Y 418.092,Z 701.938,A -85,B 0,C 180,E1 20204.354,E2 20204.354} C_VEL
LIN {X 0,Y 418.475,Z 704.927,A -85,B 0,C 180,E1 20204.046,E2 20204.046} C_VEL
LIN {X 0,Y 416.05,Z 748.273,A -85,B 0,C 180,E1 20200.092,E2 20200.092} C_VEL
LIN {X 0,Y 413.68,Z 791.84,A -85,B 0,C 180,E1 20196.136,E2 20196.136} C_VEL
LIN {X 0,Y 411.351,Z 836.879,A -85,B 0,C 180,E1 20192.077,E2 20192.077} C_VEL
LIN {X 0,Y 410.937,Z 846.126,A -85,B 0,C 180,E1 20191.278,E2 20191.278} C_VEL
LIN {X 0,Y 407.332,Z 984.97,A -85,B 0,C 180,E1 20188.138,E2 20188.138} C_VEL
LIN {X 0,Y 407.04,Z 1002.909,A -85,B 0,C 180,E1 20187.544,E2 20187.544} C_VEL
LIN {X 0,Y 406.519,Z 1019.15,A -85,B 0,C 180,E1 20186.747,E2 20186.747} C_VEL
LIN {X 0,Y 405.859,Z 1035.112,A -85,B 0,C 180,E1 20185.692,E2 20185.692} C_VEL
LIN {X 0,Y 405.033,Z 1050.712,A -85,B 0,C 180,E1 20184.343,E2 20184.343} C_VEL
LIN {X 0,Y 404.251,Z 1063.77,A -85,B 0,C 180,E1 20182.924,E2 20182.924} C_VEL
LIN {X 0,Y 403.428,Z 1076.784,A -85,B 0,C 180,E1 20181.16,E2 20181.16} C_VEL
LIN {X 0,Y 402.736,Z 1087.745,A -85,B 0,C 180,E1 20179.277,E2 20179.277} C_VEL
LIN {X 0,Y 402.248,Z 1096.696,A -85,B 0,C 180,E1 20177.351,E2 20177.351} C_VEL
LIN {X 0,Y 401.907,Z 1104.58,A -85,B 0,C 180,E1 20175.139,E2 20175.139} C_VEL
LIN {X 0,Y 401.783,Z 1109.96,A -85,B 0,C 180,E1 20173.086,E2 20173.086} C_VEL
LIN {X 0,Y 401.865,Z 1114.073,A -85,B 0,C 180,E1 20170.752,E2 20170.752} C_VEL
LIN {X 0,Y 402.157,Z 1116.057,A -85,B 0,C 180,E1 20168.576,E2 20168.576} C_VEL
LIN {X 0,Y 402.711,Z 1116.292,A -85,B 0,C 180,E1 20166.269,E2 20166.269} C_VEL
LIN {X 0,Y 403.493,Z 1114.735,A -85,B 0,C 180,E1 20164.118,E2 20164.118} C_VEL
LIN {X 0,Y 404.639,Z 1111.164,A -85,B 0,C 180,E1 20161.838,E2 20161.838} C_VEL
LIN {X 0,Y 405.936,Z 1106.251,A -85,B 0,C 180,E1 20159.84,E2 20159.84} C_VEL
LIN {X 0,Y 407.605,Z 1099.069,A -85,B 0,C 180,E1 20157.748,E2 20157.748} C_VEL
LIN {X 0,Y 409.338,Z 1090.936,A -85,B 0,C 180,E1 20155.935,E2 20155.935} C_VEL
LIN {X 0,Y 411.286,Z 1080.633,A -85,B 0,C 180,E1 20154.137,E2 20154.137} C_VEL
LIN {X 0,Y 413.176,Z 1069.202,A -85,B 0,C 180,E1 20152.558,E2 20152.558} C_VEL
LIN {X 0,Y 415.081,Z 1055.51,A -85,B 0,C 180,E1 20151.059,E2 20151.059} C_VEL
LIN {X 0,Y 416.792,Z 1040.507,A -85,B 0,C 180,E1 20149.771,E2 20149.771} C_VEL
LIN {X 0,Y 417.961,Z 1027.181,A -85,B 0,C 180,E1 20148.894,E2 20148.894} C_VEL
LIN {X 0,Y 418.837,Z 1014.286,A -85,B 0,C 180,E1 20148.22,E2 20148.22} C_VEL
LIN {X 0,Y 419.519,Z 998.86,A -85,B 0,C 180,E1 20147.615,E2 20147.615} C_VEL
LIN {X 0,Y 421.208,Z 958.138,A -85,B 0,C 180,E1 20146.532,E2 20146.532} C_VEL
LIN {X 0,Y 427.811,Z 860.53,A -85,B 0,C 180,E1 20144.023,E2 20144.023} C_VEL
LIN {X 0,Y 432.15,Z 816.896,A -85,B 0,C 180,E1 20139.972,E2 20139.972} C_VEL
LIN {X 0,Y 437.29,Z 770.81,A -85,B 0,C 180,E1 20135.693,E2 20135.693} C_VEL
LIN {X 0,Y 442.849,Z 727.625,A -85,B 0,C 180,E1 20131.657,E2 20131.657} C_VEL
LIN {X 0,Y 440.45,Z 716.812,A -85,B 0,C 180,E1 20129.734,E2 20129.734} C_VEL
LIN {X 0,Y 437.345,Z 706.869,A -85,B 0,C 180,E1 20127.521,E2 20127.521} C_VEL
LIN {X 0,Y 434.633,Z 699.696,A -85,B 0,C 180,E1 20125.442,E2 20125.442} C_VEL
LIN {X 0,Y 433.095,Z 695.894,A -85,B 0,C 180,E1 20124.095,E2 20124.095} C_VEL
LIN {X 0,Y 431.718,Z 692.339,A -85,B 0,C 180,E1 20122.596,E2 20122.596} C_VEL
LIN {X 0,Y 430.186,Z 689.028,A -85,B 0,C 180,E1 20120.611,E2 20120.611} C_VEL
LIN {X 0,Y 429.937,Z 687.917,A -85,B 0,C 180,E1 20119.916,E2 20119.916} C_VEL
LIN {X 0,Y 429.365,Z 687.402,A -85,B 0,C 180,E1 20118.878,E2 20118.878} C_VEL
LIN {X 0,Y 427.802,Z 690.117,A -85,B 0,C 180,E1 20117.806,E2 20117.806} C_VEL
LIN {X 0,Y 426.51,Z 693.098,A -85,B 0,C 180,E1 20116.797,E2 20116.797} C_VEL
LIN {X 0,Y 424.535,Z 699.523,A -85,B 0,C 180,E1 20115.562,E2 20115.562} C_VEL
LIN {X 0,Y 440.727,Z 731.878,A -85,B 0,C 180,E1 20113.114,E2 20113.114} C_VEL
LIN {X 0,Y 446.44,Z 744.332,A -85,B 0,C 180,E1 20112.277,E2 20112.277} C_VEL
LIN {X 0,Y 446.472,Z 748.647,A -85,B 0,C 180,E1 20112.159,E2 20112.159} C_VEL
LIN {X 0,Y 432.258,Z 979.23,A -85,B 0,C 180,E1 20107.194,E2 20107.194} C_VEL
LIN {X 0,Y 429.97,Z 1003.428,A -85,B 0,C 180,E1 20106.43,E2 20106.43} C_VEL
LIN {X 0,Y 427.342,Z 1025.99,A -85,B 0,C 180,E1 20105.466,E2 20105.466} C_VEL
LIN {X 0,Y 424.387,Z 1048.09,A -85,B 0,C 180,E1 20104.268,E2 20104.268} C_VEL
LIN {X 0,Y 421.061,Z 1070.273,A -85,B 0,C 180,E1 20102.778,E2 20102.778} C_VEL
LIN {X 0,Y 417.786,Z 1090.554,A -85,B 0,C 180,E1 20101.125,E2 20101.125} C_VEL
LIN {X 0,Y 414.6,Z 1109.303,A -85,B 0,C 180,E1 20099.31,E2 20099.31} C_VEL
LIN {X 0,Y 411.492,Z 1127.116,A -85,B 0,C 180,E1 20097.258,E2 20097.258} C_VEL
LIN {X 0,Y 408.634,Z 1143.432,A -85,B 0,C 180,E1 20095.041,E2 20095.041} C_VEL
LIN {X 0,Y 406.043,Z 1158.937,A -85,B 0,C 180,E1 20092.56,E2 20092.56} C_VEL
LIN {X 0,Y 404.033,Z 1171.91,A -85,B 0,C 180,E1 20090.118,E2 20090.118} C_VEL
LIN {X 0,Y 402.369,Z 1184.045,A -85,B 0,C 180,E1 20087.393,E2 20087.393} C_VEL
LIN {X 0,Y 401.248,Z 1193.887,A -85,B 0,C 180,E1 20084.723,E2 20084.723} C_VEL
LIN {X 0,Y 400.52,Z 1202.672,A -85,B 0,C 180,E1 20081.81,E2 20081.81} C_VEL
LIN {X 0,Y 400.211,Z 1209.247,A -85,B 0,C 180,E1 20079.054,E2 20079.054} C_VEL
LIN {X 0,Y 400.14,Z 1214.07,A -85,B 0,C 180,E1 20076.31,E2 20076.31} C_VEL
LIN {X 0,Y 400.17,Z 1217.441,A -85,B 0,C 180,E1 20073.579,E2 20073.579} C_VEL
LIN {X 0,Y 400.2,Z 1219.184,A -85,B 0,C 180,E1 20070.857,E2 20070.857} C_VEL
LIN {X 0,Y 400.149,Z 1219.494,A -85,B 0,C 180,E1 20067.993,E2 20067.993} C_VEL
LIN {X 0,Y 400.063,Z 1218.335,A -85,B 0,C 180,E1 20065.411,E2 20065.411} C_VEL
LIN {X 0,Y 400.054,Z 1215.379,A -85,B 0,C 180,E1 20062.386,E2 20062.386} C_VEL
LIN {X 0,Y 400.295,Z 1210.947,A -85,B 0,C 180,E1 20059.492,E2 20059.492} C_VEL
LIN {X 0,Y 400.994,Z 1204.446,A -85,B 0,C 180,E1 20056.442,E2 20056.442} C_VEL
LIN {X 0,Y 402.391,Z 1195.641,A -85,B 0,C 180,E1 20053.245,E2 20053.245} C_VEL
LIN {X 0,Y 404.378,Z 1185.761,A -85,B 0,C 180,E1 20050.348,E2 20050.348} C_VEL
LIN {X 0,Y 407.219,Z 1173.585,A -85,B 0,C 180,E1 20047.408,E2 20047.408} C_VEL
LIN {X 0,Y 410.548,Z 1160.509,A -85,B 0,C 180,E1 20044.771,E2 20044.771} C_VEL
LIN {X 0,Y 414.805,Z 1145.033,A -85,B 0,C 180,E1 20042.117,E2 20042.117} C_VEL
LIN {X 0,Y 419.673,Z 1128.11,A -85,B 0,C 180,E1 20039.66,E2 20039.66} C_VEL
LIN {X 0,Y 425.261,Z 1109.135,A -85,B 0,C 180,E1 20037.328,E2 20037.328} C_VEL
LIN {X 0,Y 431.488,Z 1088.168,A -85,B 0,C 180,E1 20035.163,E2 20035.163} C_VEL
LIN {X 0,Y 438.138,Z 1065.761,A -85,B 0,C 180,E1 20033.232,E2 20033.232} C_VEL
LIN {X 0,Y 444.949,Z 1042.618,A -85,B 0,C 180,E1 20031.584,E2 20031.584} C_VEL
LIN {X 0,Y 451.641,Z 1019.27,A -85,B 0,C 180,E1 20030.22,E2 20030.22} C_VEL
LIN {X 0,Y 458.235,Z 995.328,A -85,B 0,C 180,E1 20029.108,E2 20029.108} C_VEL
LIN {X 0,Y 465.103,Z 967.978,A -85,B 0,C 180,E1 20028.112,E2 20028.112} C_VEL
LIN {X 0,Y 484.034,Z 883.523,A -85,B 0,C 180,E1 20025.621,E2 20025.621} C_VEL
LIN {X 0,Y 492.982,Z 848.235,A -85,B 0,C 180,E1 20024.614,E2 20024.614} C_VEL
LIN {X 0,Y 475.955,Z 916.388,A -85,B 0,C 180,E1 20022.672,E2 20022.672} C_VEL
LIN {X 0,Y 466.597,Z 958.459,A -85,B 0,C 180,E1 20021.376,E2 20021.376} C_VEL
LIN {X 0,Y 460.689,Z 982.341,A -85,B 0,C 180,E1 20020.374,E2 20020.374} C_VEL
LIN {X 0,Y 454.497,Z 1005.15,A -85,B 0,C 180,E1 20019.156,E2 20019.156} C_VEL
LIN {X 0,Y 448.066,Z 1027.34,A -85,B 0,C 180,E1 20017.697,E2 20017.697} C_VEL
LIN {X 0,Y 441.56,Z 1048.741,A -85,B 0,C 180,E1 20015.991,E2 20015.991} C_VEL
LIN {X 0,Y 435.14,Z 1069.215,A -85,B 0,C 180,E1 20014.026,E2 20014.026} C_VEL
LIN {X 0,Y 429.034,Z 1088.115,A -85,B 0,C 180,E1 20011.864,E2 20011.864} C_VEL
LIN {X 0,Y 423.202,Z 1105.845,A -85,B 0,C 180,E1 20009.438,E2 20009.438} C_VEL
LIN {X 0,Y 417.871,Z 1121.88,A -85,B 0,C 180,E1 20006.806,E2 20006.806} C_VEL
LIN {X 0,Y 413.377,Z 1135.429,A -85,B 0,C 180,E1 20004.131,E2 20004.131} C_VEL
LIN {X 0,Y 409.734,Z 1146.627,A -85,B 0,C 180,E1 20001.475,E2 20001.475} C_VEL
LIN {X 0,Y 406.537,Z 1156.985,A -85,B 0,C 180,E1 19998.501,E2 19998.501} C_VEL
LIN {X 0,Y 404.223,Z 1165.054,A -85,B 0,C 180,E1 19995.645,E2 19995.645} C_VEL
LIN {X 0,Y 402.472,Z 1171.641,A -85,B 0,C 180,E1 19992.631,E2 19992.631} C_VEL
LIN {X 0,Y 401.322,Z 1176.486,A -85,B 0,C 180,E1 19989.612,E2 19989.612} C_VEL
LIN {X 0,Y 400.662,Z 1179.722,A -85,B 0,C 180,E1 19986.595,E2 19986.595} C_VEL
LIN {X 0,Y 400.339,Z 1181.258,A -85,B 0,C 180,E1 19983.726,E2 19983.726} C_VEL
LIN {X 0,Y 400.196,Z 1181.296,A -85,B 0,C 180,E1 19980.862,E2 19980.862} C_VEL
LIN {X 0,Y 400.148,Z 1179.919,A -85,B 0,C 180,E1 19977.998,E2 19977.998} C_VEL
LIN {X 0,Y 400.198,Z 1176.894,A -85,B 0,C 180,E1 19975.13,E2 19975.13} C_VEL
LIN {X 0,Y 400.428,Z 1172.076,A -85,B 0,C 180,E1 19972.109,E2 19972.109} C_VEL
LIN {X 0,Y 400.913,Z 1165.826,A -85,B 0,C 180,E1 19969.223,E2 19969.223} C_VEL
LIN {X 0,Y 401.702,Z 1158.104,A -85,B 0,C 180,E1 19966.472,E2 19966.472} C_VEL
LIN {X 0,Y 402.991,Z 1148.089,A -85,B 0,C 180,E1 19963.573,E2 19963.573} C_VEL
LIN {X 0,Y 404.627,Z 1137.247,A -85,B 0,C 180,E1 19960.966,E2 19960.966} C_VEL
LIN {X 0,Y 406.757,Z 1124.351,A -85,B 0,C 180,E1 19958.366,E2 19958.366} C_VEL
LIN {X 0,Y 409.248,Z 1109.934,A -85,B 0,C 180,E1 19955.923,E2 19955.923} C_VEL
LIN {X 0,Y 412.051,Z 1094.107,A -85,B 0,C 180,E1 19953.64,E2 19953.64} C_VEL
LIN {X 0,Y 415.112,Z 1076.827,A -85,B 0,C 180,E1 19951.519,E2 19951.519} C_VEL
LIN {X 0,Y 418.333,Z 1057.958,A -85,B 0,C 180,E1 19949.559,E2 19949.559} C_VEL
LIN {X 0,Y 421.664,Z 1037.199,A -85,B 0,C 180,E1 19947.759,E2 19947.759} C_VEL
LIN {X 0,Y 424.736,Z 1016.188,A -85,B 0,C 180,E1 19946.254,E2 19946.254} C_VEL
LIN {X 0,Y 427.427,Z 995.552,A -85,B 0,C 180,E1 19945.035,E2 19945.035} C_VEL
LIN {X 0,Y 429.977,Z 973.079,A -85,B 0,C 180,E1 19943.965,E2 19943.965} C_VEL
LIN {X 0,Y 432.076,Z 950.437,A -85,B 0,C 180,E1 19943.128,E2 19943.128} C_VEL
LIN {X 0,Y 433.788,Z 926.131,A -85,B 0,C 180,E1 19942.486,E2 19942.486} C_VEL
LIN {X 0,Y 445.84,Z 726.216,A -85,B 0,C 180,E1 19938.23,E2 19938.23} C_VEL
LIN {X 0,Y 427.551,Z 693.463,A -85,B 0,C 180,E1 19935.648,E2 19935.648} C_VEL
LIN {X 0,Y 410.133,Z 663.881,A -85,B 0,C 180,E1 19932.98,E2 19932.98} C_VEL
LIN {X 0,Y 405.239,Z 655.628,A -85,B 0,C 180,E1 19932.18,E2 19932.18} C_VEL
LIN {X 0,Y 402.993,Z 652.065,A -85,B 0,C 180,E1 19931.811,E2 19931.811} C_VEL
LIN {X 0,Y 402.63,Z 650.515,A -85,B 0,C 180,E1 19931.678,E2 19931.678} C_VEL
LIN {X 0,Y 402.629,Z 650.51,A -85,B 0,C 180,E1 19927.837,E2 19927.837} C_VEL
LIN {X 0,Y 402.661,Z 650.512,A -85,B 0,C 180,E1 19923.969,E2 19923.969} C_VEL
LIN {X 0,Y 402.672,Z 650.506,A -85,B 0,C 180,E1 19919.941,E2 19919.941} C_VEL
LIN {X 0,Y 402.641,Z 650.507,A -85,B 0,C 180,E1 19916.077,E2 19916.077} C_VEL
LIN {X 0,Y 402.593,Z 650.511,A -85,B 0,C 180,E1 19912.335,E2 19912.335} C_VEL
LIN {X 0,Y 402.615,Z 650.508,A -85,B 0,C 180,E1 19908.387,E2 19908.387} C_VEL
